# B&R Automation Studio project NAELD004C00R10L518F00 (part 9)

#### Act_OptP0200ToP0204AccDat.st
```iecst
ACTION Act_OptP0200ToP0204AccDat:

	//HComm Exchanged
	IF p_bOpsMagConvLD1HModChgDone AND p_bOpsMagConvLD2HModChgDone AND p_bOpsMagConvLD3HModChgDone THEN
		bHCommModChg := FALSE;
	END_IF

//	IF EDGENEG(p_bLFFollowerProdAccDataMnl OR p_bLCSLFAccDataMnl) THEN
//		bProdAccData	:= FALSE;
//	END_IF

	//Control
	IF (tyP0200OpsGen.tyOps.tyBtnAccDat.bRtCompl = TRUE)		OR (tyP0201OpsTravLifter.tyOps.tyBtnAccDat.bRtCompl = TRUE)
		OR (tyP0202OpsMag1.tyOps.tyBtnAccDat.bRtCompl = TRUE)	OR (tyP0203OpsMag2.tyOps.tyBtnAccDat.bRtCompl = TRUE)
		OR (tyP0204OpsMag3.tyOps.tyBtnAccDat.bRtCompl = TRUE) 	OR (tyP0206OpsMag4.tyOps.tyBtnAccDat.bRtCompl = TRUE)
		THEN

		tyP0200OpsGen.tyOps.tyBtnAccDat.bRtCompl		:= FALSE;
		tyP0201OpsTravLifter.tyOps.tyBtnAccDat.bRtCompl	:= FALSE;
		tyP0202OpsMag1.tyOps.tyBtnAccDat.bRtCompl		:= FALSE;
		tyP0203OpsMag2.tyOps.tyBtnAccDat.bRtCompl		:= FALSE;
		tyP0204OpsMag3.tyOps.tyBtnAccDat.bRtCompl		:= FALSE;
		tyP0206OpsMag4.tyOps.tyBtnAccDat.bRtCompl		:= FALSE;

		bProdAccData	:= TRUE;
	END_IF

	//Button Appearance
	IF (p_bLFFollowerProdAccDataMnl = TRUE) OR (p_bLCSLFAccDataMnl = TRUE) THEN

		fbAccDatBlinkTm(IN := TRUE);

		IF fbAccDatBlinkTm.Q THEN
			fbAccDatBlinkTm(IN := FALSE);

			IF (tyP0200OpsGen.tyOps.tyBitmapAccDat.usiValueIdx = 1) THEN
				tyP0200OpsGen.tyOps.tyBitmapAccDat.usiValueIdx			:= 0;
				tyP0201OpsTravLifter.tyOps.tyBitmapAccDat.usiValueIdx	:= 0;
				tyP0202OpsMag1.tyOps.tyBitmapAccDat.usiValueIdx			:= 0;
				tyP0203OpsMag2.tyOps.tyBitmapAccDat.usiValueIdx			:= 0;
				tyP0204OpsMag3.tyOps.tyBitmapAccDat.usiValueIdx			:= 0;
				tyP0206OpsMag4.tyOps.tyBitmapAccDat.usiValueIdx			:= 0;
			ELSE
				tyP0200OpsGen.tyOps.tyBitmapAccDat.usiValueIdx			:= 1;
				tyP0201OpsTravLifter.tyOps.tyBitmapAccDat.usiValueIdx	:= 1;
				tyP0202OpsMag1.tyOps.tyBitmapAccDat.usiValueIdx			:= 1;
				tyP0203OpsMag2.tyOps.tyBitmapAccDat.usiValueIdx			:= 1;
				tyP0204OpsMag3.tyOps.tyBitmapAccDat.usiValueIdx			:= 1;
				tyP0206OpsMag4.tyOps.tyBitmapAccDat.usiValueIdx			:= 1;
			END_IF
		END_IF

		fUIInRtStatOff(ADR(tyP0200OpsGen.tyOps.tyBtnAccDat.uiRtStat));
		fUIInRtStatOff(ADR(tyP0201OpsTravLifter.tyOps.tyBtnAccDat.uiRtStat));
		fUIInRtStatOff(ADR(tyP0202OpsMag1.tyOps.tyBtnAccDat.uiRtStat));
		fUIInRtStatOff(ADR(tyP0203OpsMag2.tyOps.tyBtnAccDat.uiRtStat));
		fUIInRtStatOff(ADR(tyP0204OpsMag3.tyOps.tyBtnAccDat.uiRtStat));
		fUIInRtStatOff(ADR(tyP0206OpsMag4.tyOps.tyBtnAccDat.uiRtStat));

		fUIInRtStatOff(ADR(tyP0200OpsGen.tyOps.tyBitmapAccDat.uiRtStat));
		fUIInRtStatOff(ADR(tyP0201OpsTravLifter.tyOps.tyBitmapAccDat.uiRtStat));
		fUIInRtStatOff(ADR(tyP0202OpsMag1.tyOps.tyBitmapAccDat.uiRtStat));
		fUIInRtStatOff(ADR(tyP0203OpsMag2.tyOps.tyBitmapAccDat.uiRtStat));
		fUIInRtStatOff(ADR(tyP0204OpsMag3.tyOps.tyBitmapAccDat.uiRtStat));
		fUIInRtStatOff(ADR(tyP0206OpsMag4.tyOps.tyBitmapAccDat.uiRtStat));
	ELSE

		fbAccDatBlinkTm(IN := FALSE);

		tyP0200OpsGen.tyOps.tyBitmapAccDat.usiValueIdx			:= 0;
		tyP0201OpsTravLifter.tyOps.tyBitmapAccDat.usiValueIdx	:= 0;
		tyP0202OpsMag1.tyOps.tyBitmapAccDat.usiValueIdx			:= 0;
		tyP0203OpsMag2.tyOps.tyBitmapAccDat.usiValueIdx			:= 0;
		tyP0204OpsMag3.tyOps.tyBitmapAccDat.usiValueIdx			:= 0;
		tyP0206OpsMag4.tyOps.tyBitmapAccDat.usiValueIdx			:= 0;

		fUIInRtStatHide(ADR(tyP0200OpsGen.tyOps.tyBtnAccDat.uiRtStat));
		fUIInRtStatHide(ADR(tyP0201OpsTravLifter.tyOps.tyBtnAccDat.uiRtStat));
		fUIInRtStatHide(ADR(tyP0202OpsMag1.tyOps.tyBtnAccDat.uiRtStat));
		fUIInRtStatHide(ADR(tyP0203OpsMag2.tyOps.tyBtnAccDat.uiRtStat));
		fUIInRtStatHide(ADR(tyP0204OpsMag3.tyOps.tyBtnAccDat.uiRtStat));
		fUIInRtStatHide(ADR(tyP0206OpsMag4.tyOps.tyBtnAccDat.uiRtStat));

		fUIInRtStatHide(ADR(tyP0200OpsGen.tyOps.tyBitmapAccDat.uiRtStat));
		fUIInRtStatHide(ADR(tyP0201OpsTravLifter.tyOps.tyBitmapAccDat.uiRtStat));
		fUIInRtStatHide(ADR(tyP0202OpsMag1.tyOps.tyBitmapAccDat.uiRtStat));
		fUIInRtStatHide(ADR(tyP0203OpsMag2.tyOps.tyBitmapAccDat.uiRtStat));
		fUIInRtStatHide(ADR(tyP0204OpsMag3.tyOps.tyBitmapAccDat.uiRtStat));
		fUIInRtStatHide(ADR(tyP0206OpsMag4.tyOps.tyBitmapAccDat.uiRtStat));
	END_IF

//	IF p_tyNtParamCurr.bLFPrep AND p_tyMcParamCurr.bLFEn THEN
//		IF p_bLFFollowerDSAllow=FALSE THEN
//			tyP0200OpsGen.tyOps.tyTxtLdrInActiveCtrl.usiValueIdx	:= 0;
//			tyP0201OpsTravLifter.tyOps.tyTxtLdrInActiveCtrl.usiValueIdx	:= 0;
//			tyP0202OpsMag1.tyOps.tyTxtLdrInActiveCtrl.usiValueIdx	:= 0;
//			tyP0203OpsMag2.tyOps.tyTxtLdrInActiveCtrl.usiValueIdx	:= 0;
//			tyP0204OpsMag3.tyOps.tyTxtLdrInActiveCtrl.usiValueIdx	:= 0;
//
//			fUIInRtStatOff(ADR(tyP0200OpsGen.tyOps.tyTxtLdrInActiveCtrl.uiRtStat));
//			fUIInRtStatOff(ADR(tyP0201OpsTravLifter.tyOps.tyTxtLdrInActiveCtrl.uiRtStat));
//			fUIInRtStatOff(ADR(tyP0202OpsMag1.tyOps.tyTxtLdrInActiveCtrl.uiRtStat));
//			fUIInRtStatOff(ADR(tyP0203OpsMag2.tyOps.tyTxtLdrInActiveCtrl.uiRtStat));
//			fUIInRtStatOff(ADR(tyP0204OpsMag3.tyOps.tyTxtLdrInActiveCtrl.uiRtStat));
//
//			fUIInRtStatOff(ADR(tyP0200OpsGen.tyOps.tyBitmapWarningLF.uiRtStat));
//			fUIInRtStatOff(ADR(tyP0201OpsTravLifter.tyOps.tyBitmapWarningLF.uiRtStat));
//			fUIInRtStatOff(ADR(tyP0202OpsMag1.tyOps.tyBitmapWarningLF.uiRtStat));
//			fUIInRtStatOff(ADR(tyP0203OpsMag2.tyOps.tyBitmapWarningLF.uiRtStat));
//			fUIInRtStatOff(ADR(tyP0204OpsMag3.tyOps.tyBitmapWarningLF.uiRtStat));
//
//		ELSIF p_bLFFollowerUSAllow=FALSE THEN
//			IF p_tyMcParamCurr.bSectionLeader THEN
//				tyP0200OpsGen.tyOps.tyTxtLdrInActiveCtrl.usiValueIdx	:= 3;
//				tyP0201OpsTravLifter.tyOps.tyTxtLdrInActiveCtrl.usiValueIdx	:= 3;
//				tyP0202OpsMag1.tyOps.tyTxtLdrInActiveCtrl.usiValueIdx	:= 3;
//				tyP0203OpsMag2.tyOps.tyTxtLdrInActiveCtrl.usiValueIdx	:= 3;
//				tyP0204OpsMag3.tyOps.tyTxtLdrInActiveCtrl.usiValueIdx	:= 3;
//
//				fUIInRtStatOff(ADR(tyP0200OpsGen.tyOps.tyTxtLdrInActiveCtrl.uiRtStat));
//				fUIInRtStatOff(ADR(tyP0201OpsTravLifter.tyOps.tyTxtLdrInActiveCtrl.uiRtStat));
//				fUIInRtStatOff(ADR(tyP0202OpsMag1.tyOps.tyTxtLdrInActiveCtrl.uiRtStat));
//				fUIInRtStatOff(ADR(tyP0203OpsMag2.tyOps.tyTxtLdrInActiveCtrl.uiRtStat));
//				fUIInRtStatOff(ADR(tyP0204OpsMag3.tyOps.tyTxtLdrInActiveCtrl.uiRtStat));
//
//				fUIInRtStatOff(ADR(tyP0200OpsGen.tyOps.tyBitmapWarningLF.uiRtStat));
//				fUIInRtStatOff(ADR(tyP0201OpsTravLifter.tyOps.tyBitmapWarningLF.uiRtStat));
//				fUIInRtStatOff(ADR(tyP0202OpsMag1.tyOps.tyBitmapWarningLF.uiRtStat));
//				fUIInRtStatOff(ADR(tyP0203OpsMag2.tyOps.tyBitmapWarningLF.uiRtStat));
//				fUIInRtStatOff(ADR(tyP0204OpsMag3.tyOps.tyBitmapWarningLF.uiRtStat));
//			ELSE
//				tyP0200OpsGen.tyOps.tyTxtLdrInActiveCtrl.usiValueIdx	:= 2;
//				tyP0201OpsTravLifter.tyOps.tyTxtLdrInActiveCtrl.usiValueIdx	:= 2;
//				tyP0202OpsMag1.tyOps.tyTxtLdrInActiveCtrl.usiValueIdx	:= 2;
//				tyP0203OpsMag2.tyOps.tyTxtLdrInActiveCtrl.usiValueIdx	:= 2;
//				tyP0204OpsMag3.tyOps.tyTxtLdrInActiveCtrl.usiValueIdx	:= 2;
//
//				fUIInRtStatOff(ADR(tyP0200OpsGen.tyOps.tyTxtLdrInActiveCtrl.uiRtStat));
//				fUIInRtStatOff(ADR(tyP0201OpsTravLifter.tyOps.tyTxtLdrInActiveCtrl.uiRtStat));
//				fUIInRtStatOff(ADR(tyP0202OpsMag1.tyOps.tyTxtLdrInActiveCtrl.uiRtStat));
//				fUIInRtStatOff(ADR(tyP0203OpsMag2.tyOps.tyTxtLdrInActiveCtrl.uiRtStat));
//				fUIInRtStatOff(ADR(tyP0204OpsMag3.tyOps.tyTxtLdrInActiveCtrl.uiRtStat));
//
//				fUIInRtStatOff(ADR(tyP0200OpsGen.tyOps.tyBitmapWarningLF.uiRtStat));
//				fUIInRtStatOff(ADR(tyP0201OpsTravLifter.tyOps.tyBitmapWarningLF.uiRtStat));
//				fUIInRtStatOff(ADR(tyP0202OpsMag1.tyOps.tyBitmapWarningLF.uiRtStat));
//				fUIInRtStatOff(ADR(tyP0203OpsMag2.tyOps.tyBitmapWarningLF.uiRtStat));
//				fUIInRtStatOff(ADR(tyP0204OpsMag3.tyOps.tyBitmapWarningLF.uiRtStat));
//			END_IF
//		ELSE
//			IF p_bLFFollowerLdrSeqCtrlInActive THEN
//				tyP0200OpsGen.tyOps.tyTxtLdrInActiveCtrl.usiValueIdx	:= 1;
//				tyP0201OpsTravLifter.tyOps.tyTxtLdrInActiveCtrl.usiValueIdx	:= 1;
//				tyP0202OpsMag1.tyOps.tyTxtLdrInActiveCtrl.usiValueIdx	:= 1;
//				tyP0203OpsMag2.tyOps.tyTxtLdrInActiveCtrl.usiValueIdx	:= 1;
//				tyP0204OpsMag3.tyOps.tyTxtLdrInActiveCtrl.usiValueIdx	:= 1;
//
//				fUIInRtStatOff(ADR(tyP0200OpsGen.tyOps.tyTxtLdrInActiveCtrl.uiRtStat));
//				fUIInRtStatOff(ADR(tyP0201OpsTravLifter.tyOps.tyTxtLdrInActiveCtrl.uiRtStat));
//				fUIInRtStatOff(ADR(tyP0202OpsMag1.tyOps.tyTxtLdrInActiveCtrl.uiRtStat));
//				fUIInRtStatOff(ADR(tyP0203OpsMag2.tyOps.tyTxtLdrInActiveCtrl.uiRtStat));
//				fUIInRtStatOff(ADR(tyP0204OpsMag3.tyOps.tyTxtLdrInActiveCtrl.uiRtStat));
//
//				fUIInRtStatOff(ADR(tyP0200OpsGen.tyOps.tyBitmapWarningLF.uiRtStat));
//				fUIInRtStatOff(ADR(tyP0201OpsTravLifter.tyOps.tyBitmapWarningLF.uiRtStat));
//				fUIInRtStatOff(ADR(tyP0202OpsMag1.tyOps.tyBitmapWarningLF.uiRtStat));
//				fUIInRtStatOff(ADR(tyP0203OpsMag2.tyOps.tyBitmapWarningLF.uiRtStat));
//				fUIInRtStatOff(ADR(tyP0204OpsMag3.tyOps.tyBitmapWarningLF.uiRtStat));
//			ELSE
//				fUIInRtStatHide(ADR(tyP0200OpsGen.tyOps.tyTxtLdrInActiveCtrl.uiRtStat));
//				fUIInRtStatHide(ADR(tyP0201OpsTravLifter.tyOps.tyTxtLdrInActiveCtrl.uiRtStat));
//				fUIInRtStatHide(ADR(tyP0202OpsMag1.tyOps.tyTxtLdrInActiveCtrl.uiRtStat));
//				fUIInRtStatHide(ADR(tyP0203OpsMag2.tyOps.tyTxtLdrInActiveCtrl.uiRtStat));
//				fUIInRtStatHide(ADR(tyP0204OpsMag3.tyOps.tyTxtLdrInActiveCtrl.uiRtStat));
//
//				fUIInRtStatHide(ADR(tyP0200OpsGen.tyOps.tyBitmapWarningLF.uiRtStat));
//				fUIInRtStatHide(ADR(tyP0201OpsTravLifter.tyOps.tyBitmapWarningLF.uiRtStat));
//				fUIInRtStatHide(ADR(tyP0202OpsMag1.tyOps.tyBitmapWarningLF.uiRtStat));
//				fUIInRtStatHide(ADR(tyP0203OpsMag2.tyOps.tyBitmapWarningLF.uiRtStat));
//				fUIInRtStatHide(ADR(tyP0204OpsMag3.tyOps.tyBitmapWarningLF.uiRtStat));
//			END_IF
//		END_IF
//	ELSE
//		fUIInRtStatHide(ADR(tyP0200OpsGen.tyOps.tyTxtLdrInActiveCtrl.uiRtStat));
//		fUIInRtStatHide(ADR(tyP0201OpsTravLifter.tyOps.tyTxtLdrInActiveCtrl.uiRtStat));
//		fUIInRtStatHide(ADR(tyP0202OpsMag1.tyOps.tyTxtLdrInActiveCtrl.uiRtStat));
//		fUIInRtStatHide(ADR(tyP0203OpsMag2.tyOps.tyTxtLdrInActiveCtrl.uiRtStat));
//		fUIInRtStatHide(ADR(tyP0204OpsMag3.tyOps.tyTxtLdrInActiveCtrl.uiRtStat));
//
//		fUIInRtStatHide(ADR(tyP0200OpsGen.tyOps.tyBitmapWarningLF.uiRtStat));
//		fUIInRtStatHide(ADR(tyP0201OpsTravLifter.tyOps.tyBitmapWarningLF.uiRtStat));
//		fUIInRtStatHide(ADR(tyP0202OpsMag1.tyOps.tyBitmapWarningLF.uiRtStat));
//		fUIInRtStatHide(ADR(tyP0203OpsMag2.tyOps.tyBitmapWarningLF.uiRtStat));
//		fUIInRtStatHide(ADR(tyP0204OpsMag3.tyOps.tyBitmapWarningLF.uiRtStat));
//	END_IF

END_ACTION
```

#### Act_OptP0200ToP0204BypsInitConv.st
```iecst
ACTION Act_OptP0200ToP0204BypsInitConv:

	IF p_tyNtParamCurr.bProjBypsInitConvPrep THEN

		(*Display*)
		//Initializing Conveyor
		IF EDGEPOS(p_bOpsTravLifLDInitConv) THEN
			fUIInRtStatOff(ADR(tyP0200OpsGen.tyBypsInitConv.tyLyr.uiRtStat));
			fUIInRtStatOff(ADR(tyP0201OpsTravLifter.tyBypsInitConv.tyLyr.uiRtStat));
			fUIInRtStatOff(ADR(tyP0202OpsMag1.tyBypsInitConv.tyLyr.uiRtStat));
			fUIInRtStatOff(ADR(tyP0203OpsMag2.tyBypsInitConv.tyLyr.uiRtStat));
			fUIInRtStatOff(ADR(tyP0204OpsMag3.tyBypsInitConv.tyLyr.uiRtStat));
			fUIInRtStatOff(ADR(tyP0206OpsMag4.tyBypsInitConv.tyLyr.uiRtStat));
		END_IF

		//Initializing Conveyor Done
		IF EDGENEG(p_bOpsTravLifLDInitConv) THEN
			fUIInRtStatHide(ADR(tyP0200OpsGen.tyBypsInitConv.tyLyr.uiRtStat));
			fUIInRtStatHide(ADR(tyP0201OpsTravLifter.tyBypsInitConv.tyLyr.uiRtStat));
			fUIInRtStatHide(ADR(tyP0202OpsMag1.tyBypsInitConv.tyLyr.uiRtStat));
			fUIInRtStatHide(ADR(tyP0203OpsMag2.tyBypsInitConv.tyLyr.uiRtStat));
			fUIInRtStatHide(ADR(tyP0204OpsMag3.tyBypsInitConv.tyLyr.uiRtStat));
			fUIInRtStatHide(ADR(tyP0206OpsMag4.tyBypsInitConv.tyLyr.uiRtStat));

			bOpsBypsInitConv	:= FALSE;
		END_IF

		//Blinking Button
		IF tyP0200OpsGen.tyBypsInitConv.tyLyr.uiRtStat.0 = FALSE THEN

			fbBypsInitConvBlinkTm(IN := TRUE);

			IF fbBypsInitConvBlinkTm.Q THEN
				fbBypsInitConvBlinkTm(IN := FALSE);

				IF tyP0200OpsGen.tyBypsInitConv.tyBtnBypsInitConv.usiBitmapIdx = 0 THEN
					tyP0200OpsGen.tyBypsInitConv.tyBtnBypsInitConv.usiBitmapIdx			:= 1;
					tyP0201OpsTravLifter.tyBypsInitConv.tyBtnBypsInitConv.usiBitmapIdx	:= 1;
					tyP0202OpsMag1.tyBypsInitConv.tyBtnBypsInitConv.usiBitmapIdx		:= 1;
					tyP0203OpsMag2.tyBypsInitConv.tyBtnBypsInitConv.usiBitmapIdx		:= 1;
					tyP0204OpsMag3.tyBypsInitConv.tyBtnBypsInitConv.usiBitmapIdx		:= 1;
					tyP0206OpsMag4.tyBypsInitConv.tyBtnBypsInitConv.usiBitmapIdx		:= 1;
				ELSE
					tyP0200OpsGen.tyBypsInitConv.tyBtnBypsInitConv.usiBitmapIdx			:= 0;
					tyP0201OpsTravLifter.tyBypsInitConv.tyBtnBypsInitConv.usiBitmapIdx	:= 0;
					tyP0202OpsMag1.tyBypsInitConv.tyBtnBypsInitConv.usiBitmapIdx		:= 0;
					tyP0203OpsMag2.tyBypsInitConv.tyBtnBypsInitConv.usiBitmapIdx		:= 0;
					tyP0204OpsMag3.tyBypsInitConv.tyBtnBypsInitConv.usiBitmapIdx		:= 0;
					tyP0206OpsMag4.tyBypsInitConv.tyBtnBypsInitConv.usiBitmapIdx		:= 0;
				END_IF

			END_IF

		ELSE

			fbBypsInitConvBlinkTm(IN := FALSE);

			tyP0200OpsGen.tyBypsInitConv.tyBtnBypsInitConv.usiBitmapIdx			:= 0;
			tyP0201OpsTravLifter.tyBypsInitConv.tyBtnBypsInitConv.usiBitmapIdx	:= 0;
			tyP0202OpsMag1.tyBypsInitConv.tyBtnBypsInitConv.usiBitmapIdx		:= 0;
			tyP0203OpsMag2.tyBypsInitConv.tyBtnBypsInitConv.usiBitmapIdx		:= 0;
			tyP0204OpsMag3.tyBypsInitConv.tyBtnBypsInitConv.usiBitmapIdx		:= 0;
			tyP0206OpsMag4.tyBypsInitConv.tyBtnBypsInitConv.usiBitmapIdx		:= 0;
		END_IF

		(*Control*)
		IF tyP0200OpsGen.tyBypsInitConv.tyBtnBypsInitConv.bRtCompl
			OR tyP0201OpsTravLifter.tyBypsInitConv.tyBtnBypsInitConv.bRtCompl
			OR tyP0202OpsMag1.tyBypsInitConv.tyBtnBypsInitConv.bRtCompl
			OR tyP0203OpsMag2.tyBypsInitConv.tyBtnBypsInitConv.bRtCompl
			OR tyP0204OpsMag3.tyBypsInitConv.tyBtnBypsInitConv.bRtCompl
			OR tyP0206OpsMag4.tyBypsInitConv.tyBtnBypsInitConv.bRtCompl
			THEN
			tyP0200OpsGen.tyBypsInitConv.tyBtnBypsInitConv.bRtCompl			:= FALSE;
			tyP0201OpsTravLifter.tyBypsInitConv.tyBtnBypsInitConv.bRtCompl	:= FALSE;
			tyP0202OpsMag1.tyBypsInitConv.tyBtnBypsInitConv.bRtCompl		:= FALSE;
			tyP0203OpsMag2.tyBypsInitConv.tyBtnBypsInitConv.bRtCompl		:= FALSE;
			tyP0204OpsMag3.tyBypsInitConv.tyBtnBypsInitConv.bRtCompl		:= FALSE;
			tyP0206OpsMag4.tyBypsInitConv.tyBtnBypsInitConv.bRtCompl		:= FALSE;

			fUIInRtStatHide(ADR(tyP0200OpsGen.tyBypsInitConv.tyLyr.uiRtStat));
			fUIInRtStatHide(ADR(tyP0201OpsTravLifter.tyBypsInitConv.tyLyr.uiRtStat));
			fUIInRtStatHide(ADR(tyP0202OpsMag1.tyBypsInitConv.tyLyr.uiRtStat));
			fUIInRtStatHide(ADR(tyP0203OpsMag2.tyBypsInitConv.tyLyr.uiRtStat));
			fUIInRtStatHide(ADR(tyP0204OpsMag3.tyBypsInitConv.tyLyr.uiRtStat));
			fUIInRtStatHide(ADR(tyP0206OpsMag4.tyBypsInitConv.tyLyr.uiRtStat));
			bOpsBypsInitConv	:= TRUE;

		ELSIF tyP0200OpsGen.tyBypsInitConv.tyHotspotClose.bRtCompl
			OR tyP0201OpsTravLifter.tyBypsInitConv.tyHotspotClose.bRtCompl
			OR tyP0202OpsMag1.tyBypsInitConv.tyHotspotClose.bRtCompl
			OR tyP0203OpsMag2.tyBypsInitConv.tyHotspotClose.bRtCompl
			OR tyP0204OpsMag3.tyBypsInitConv.tyHotspotClose.bRtCompl
			OR tyP0206OpsMag4.tyBypsInitConv.tyHotspotClose.bRtCompl
			THEN
			tyP0200OpsGen.tyBypsInitConv.tyHotspotClose.bRtCompl		:= FALSE;
			tyP0201OpsTravLifter.tyBypsInitConv.tyHotspotClose.bRtCompl	:= FALSE;
			tyP0202OpsMag1.tyBypsInitConv.tyHotspotClose.bRtCompl		:= FALSE;
			tyP0203OpsMag2.tyBypsInitConv.tyHotspotClose.bRtCompl		:= FALSE;
			tyP0204OpsMag3.tyBypsInitConv.tyHotspotClose.bRtCompl		:= FALSE;
			tyP0206OpsMag4.tyBypsInitConv.tyHotspotClose.bRtCompl		:= FALSE;

			fUIInRtStatHide(ADR(tyP0200OpsGen.tyBypsInitConv.tyLyr.uiRtStat));
			fUIInRtStatHide(ADR(tyP0201OpsTravLifter.tyBypsInitConv.tyLyr.uiRtStat));
			fUIInRtStatHide(ADR(tyP0202OpsMag1.tyBypsInitConv.tyLyr.uiRtStat));
			fUIInRtStatHide(ADR(tyP0203OpsMag2.tyBypsInitConv.tyLyr.uiRtStat));
			fUIInRtStatHide(ADR(tyP0204OpsMag3.tyBypsInitConv.tyLyr.uiRtStat));
			fUIInRtStatHide(ADR(tyP0206OpsMag4.tyBypsInitConv.tyLyr.uiRtStat));
		END_IF

	END_IF

END_ACTION
```

#### Act_OptP0200ToP0204_P0003AccDat.st - not listed in the package file held
```iecst
ACTION Act_OptP0200ToP0204_P0003AccDat:

	//HComm Exchanged
	IF p_bOpsMagConvLD1HModChgDone AND p_bOpsMagConvLD2HModChgDone AND p_bOpsMagConvLD3HModChgDone THEN
		bHCommModChg := FALSE;
	END_IF

//	IF EDGENEG(p_bLFFollowerProdAccDataMnl OR p_bLCSLFAccDataMnl) THEN
//		bProdAccData	:= FALSE;
//	END_IF

	//Control
	IF (tyP0200OpsGen.tyOps.tyBtnAccDat.bRtCompl = TRUE)		OR (tyP0201OpsTravLifter.tyOps.tyBtnAccDat.bRtCompl = TRUE)
		OR (tyP0202OpsMag1.tyOps.tyBtnAccDat.bRtCompl = TRUE)	OR (tyP0203OpsMag2.tyOps.tyBtnAccDat.bRtCompl = TRUE)
		OR (tyP0204OpsMag3.tyOps.tyBtnAccDat.bRtCompl = TRUE) 	OR (tyP0206OpsMag4.tyOps.tyBtnAccDat.bRtCompl = TRUE)
		OR tyP0003MMenu.tyMMenuBtn.tyBtnAccDat.bRtCompl THEN

		tyP0200OpsGen.tyOps.tyBtnAccDat.bRtCompl		:= FALSE;
		tyP0201OpsTravLifter.tyOps.tyBtnAccDat.bRtCompl	:= FALSE;
		tyP0202OpsMag1.tyOps.tyBtnAccDat.bRtCompl		:= FALSE;
		tyP0203OpsMag2.tyOps.tyBtnAccDat.bRtCompl		:= FALSE;
		tyP0204OpsMag3.tyOps.tyBtnAccDat.bRtCompl		:= FALSE;
		tyP0206OpsMag4.tyOps.tyBtnAccDat.bRtCompl		:= FALSE;
		tyP0003MMenu.tyMMenuBtn.tyBtnAccDat.bRtCompl := FALSE;

		bProdAccData	:= TRUE;
	END_IF

	//Button Appearance
	IF (p_bLFFollowerProdAccDataMnl = TRUE) OR (p_bLCSLFAccDataMnl = TRUE) THEN

		fbAccDatBlinkTm(IN := TRUE);

		IF fbAccDatBlinkTm.Q THEN
			fbAccDatBlinkTm(IN := FALSE);

			IF (tyP0200OpsGen.tyOps.tyBitmapAccDat.usiValueIdx = 1) THEN
				tyP0200OpsGen.tyOps.tyBitmapAccDat.usiValueIdx			:= 0;
				tyP0201OpsTravLifter.tyOps.tyBitmapAccDat.usiValueIdx	:= 0;
				tyP0202OpsMag1.tyOps.tyBitmapAccDat.usiValueIdx			:= 0;
				tyP0203OpsMag2.tyOps.tyBitmapAccDat.usiValueIdx			:= 0;
				tyP0204OpsMag3.tyOps.tyBitmapAccDat.usiValueIdx			:= 0;
				tyP0206OpsMag4.tyOps.tyBitmapAccDat.usiValueIdx			:= 0;
				tyP0003MMenu.tyMMenuBtn.tyBtnAccDat.usiBitmapIdx := 0;
			ELSE
				tyP0200OpsGen.tyOps.tyBitmapAccDat.usiValueIdx			:= 1;
				tyP0201OpsTravLifter.tyOps.tyBitmapAccDat.usiValueIdx	:= 1;
				tyP0202OpsMag1.tyOps.tyBitmapAccDat.usiValueIdx			:= 1;
				tyP0203OpsMag2.tyOps.tyBitmapAccDat.usiValueIdx			:= 1;
				tyP0204OpsMag3.tyOps.tyBitmapAccDat.usiValueIdx			:= 1;
				tyP0206OpsMag4.tyOps.tyBitmapAccDat.usiValueIdx			:= 1;
				tyP0003MMenu.tyMMenuBtn.tyBtnAccDat.usiBitmapIdx := 4;
			END_IF
		END_IF

		fUIInRtStatOff(ADR(tyP0200OpsGen.tyOps.tyBtnAccDat.uiRtStat));
		fUIInRtStatOff(ADR(tyP0201OpsTravLifter.tyOps.tyBtnAccDat.uiRtStat));
		fUIInRtStatOff(ADR(tyP0202OpsMag1.tyOps.tyBtnAccDat.uiRtStat));
		fUIInRtStatOff(ADR(tyP0203OpsMag2.tyOps.tyBtnAccDat.uiRtStat));
		fUIInRtStatOff(ADR(tyP0204OpsMag3.tyOps.tyBtnAccDat.uiRtStat));
		fUIInRtStatOff(ADR(tyP0206OpsMag4.tyOps.tyBtnAccDat.uiRtStat));

		fUIInRtStatOff(ADR(tyP0200OpsGen.tyOps.tyBitmapAccDat.uiRtStat));
		fUIInRtStatOff(ADR(tyP0201OpsTravLifter.tyOps.tyBitmapAccDat.uiRtStat));
		fUIInRtStatOff(ADR(tyP0202OpsMag1.tyOps.tyBitmapAccDat.uiRtStat));
		fUIInRtStatOff(ADR(tyP0203OpsMag2.tyOps.tyBitmapAccDat.uiRtStat));
		fUIInRtStatOff(ADR(tyP0204OpsMag3.tyOps.tyBitmapAccDat.uiRtStat));
		fUIInRtStatOff(ADR(tyP0206OpsMag4.tyOps.tyBitmapAccDat.uiRtStat));

		fUIInRtStatOff(ADR(tyP0003MMenu.tyMMenuBtn.tyBtnAccDat.uiRtStat));
	ELSE

		fbAccDatBlinkTm(IN := FALSE);

		tyP0200OpsGen.tyOps.tyBitmapAccDat.usiValueIdx			:= 0;
		tyP0201OpsTravLifter.tyOps.tyBitmapAccDat.usiValueIdx	:= 0;
		tyP0202OpsMag1.tyOps.tyBitmapAccDat.usiValueIdx			:= 0;
		tyP0203OpsMag2.tyOps.tyBitmapAccDat.usiValueIdx			:= 0;
		tyP0204OpsMag3.tyOps.tyBitmapAccDat.usiValueIdx			:= 0;
		tyP0206OpsMag4.tyOps.tyBitmapAccDat.usiValueIdx			:= 0;

		fUIInRtStatHide(ADR(tyP0200OpsGen.tyOps.tyBtnAccDat.uiRtStat));
		fUIInRtStatHide(ADR(tyP0201OpsTravLifter.tyOps.tyBtnAccDat.uiRtStat));
		fUIInRtStatHide(ADR(tyP0202OpsMag1.tyOps.tyBtnAccDat.uiRtStat));
		fUIInRtStatHide(ADR(tyP0203OpsMag2.tyOps.tyBtnAccDat.uiRtStat));
		fUIInRtStatHide(ADR(tyP0204OpsMag3.tyOps.tyBtnAccDat.uiRtStat));
		fUIInRtStatHide(ADR(tyP0206OpsMag4.tyOps.tyBtnAccDat.uiRtStat));

		fUIInRtStatHide(ADR(tyP0200OpsGen.tyOps.tyBitmapAccDat.uiRtStat));
		fUIInRtStatHide(ADR(tyP0201OpsTravLifter.tyOps.tyBitmapAccDat.uiRtStat));
		fUIInRtStatHide(ADR(tyP0202OpsMag1.tyOps.tyBitmapAccDat.uiRtStat));
		fUIInRtStatHide(ADR(tyP0203OpsMag2.tyOps.tyBitmapAccDat.uiRtStat));
		fUIInRtStatHide(ADR(tyP0204OpsMag3.tyOps.tyBitmapAccDat.uiRtStat));
		fUIInRtStatHide(ADR(tyP0206OpsMag4.tyOps.tyBitmapAccDat.uiRtStat));

		fUIInRtStatHide(ADR(tyP0003MMenu.tyMMenuBtn.tyBtnAccDat.uiRtStat));
	END_IF

//	IF p_tyNtParamCurr.bLFPrep AND p_tyMcParamCurr.bLFEn THEN
//		IF p_bLFFollowerDSAllow=FALSE THEN
//			tyP0200OpsGen.tyOps.tyTxtLdrInActiveCtrl.usiValueIdx	:= 0;
//			tyP0201OpsTravLifter.tyOps.tyTxtLdrInActiveCtrl.usiValueIdx	:= 0;
//			tyP0202OpsMag1.tyOps.tyTxtLdrInActiveCtrl.usiValueIdx	:= 0;
//			tyP0203OpsMag2.tyOps.tyTxtLdrInActiveCtrl.usiValueIdx	:= 0;
//			tyP0204OpsMag3.tyOps.tyTxtLdrInActiveCtrl.usiValueIdx	:= 0;
//
//			fUIInRtStatOff(ADR(tyP0200OpsGen.tyOps.tyTxtLdrInActiveCtrl.uiRtStat));
//			fUIInRtStatOff(ADR(tyP0201OpsTravLifter.tyOps.tyTxtLdrInActiveCtrl.uiRtStat));
//			fUIInRtStatOff(ADR(tyP0202OpsMag1.tyOps.tyTxtLdrInActiveCtrl.uiRtStat));
//			fUIInRtStatOff(ADR(tyP0203OpsMag2.tyOps.tyTxtLdrInActiveCtrl.uiRtStat));
//			fUIInRtStatOff(ADR(tyP0204OpsMag3.tyOps.tyTxtLdrInActiveCtrl.uiRtStat));
//
//			fUIInRtStatOff(ADR(tyP0200OpsGen.tyOps.tyBitmapWarningLF.uiRtStat));
//			fUIInRtStatOff(ADR(tyP0201OpsTravLifter.tyOps.tyBitmapWarningLF.uiRtStat));
//			fUIInRtStatOff(ADR(tyP0202OpsMag1.tyOps.tyBitmapWarningLF.uiRtStat));
//			fUIInRtStatOff(ADR(tyP0203OpsMag2.tyOps.tyBitmapWarningLF.uiRtStat));
//			fUIInRtStatOff(ADR(tyP0204OpsMag3.tyOps.tyBitmapWarningLF.uiRtStat));
//
//		ELSIF p_bLFFollowerUSAllow=FALSE THEN
//			IF p_tyMcParamCurr.bSectionLeader THEN
//				tyP0200OpsGen.tyOps.tyTxtLdrInActiveCtrl.usiValueIdx	:= 3;
//				tyP0201OpsTravLifter.tyOps.tyTxtLdrInActiveCtrl.usiValueIdx	:= 3;
//				tyP0202OpsMag1.tyOps.tyTxtLdrInActiveCtrl.usiValueIdx	:= 3;
//				tyP0203OpsMag2.tyOps.tyTxtLdrInActiveCtrl.usiValueIdx	:= 3;
//				tyP0204OpsMag3.tyOps.tyTxtLdrInActiveCtrl.usiValueIdx	:= 3;
//
//				fUIInRtStatOff(ADR(tyP0200OpsGen.tyOps.tyTxtLdrInActiveCtrl.uiRtStat));
//				fUIInRtStatOff(ADR(tyP0201OpsTravLifter.tyOps.tyTxtLdrInActiveCtrl.uiRtStat));
//				fUIInRtStatOff(ADR(tyP0202OpsMag1.tyOps.tyTxtLdrInActiveCtrl.uiRtStat));
//				fUIInRtStatOff(ADR(tyP0203OpsMag2.tyOps.tyTxtLdrInActiveCtrl.uiRtStat));
//				fUIInRtStatOff(ADR(tyP0204OpsMag3.tyOps.tyTxtLdrInActiveCtrl.uiRtStat));
//
//				fUIInRtStatOff(ADR(tyP0200OpsGen.tyOps.tyBitmapWarningLF.uiRtStat));
//				fUIInRtStatOff(ADR(tyP0201OpsTravLifter.tyOps.tyBitmapWarningLF.uiRtStat));
//				fUIInRtStatOff(ADR(tyP0202OpsMag1.tyOps.tyBitmapWarningLF.uiRtStat));
//				fUIInRtStatOff(ADR(tyP0203OpsMag2.tyOps.tyBitmapWarningLF.uiRtStat));
//				fUIInRtStatOff(ADR(tyP0204OpsMag3.tyOps.tyBitmapWarningLF.uiRtStat));
//			ELSE
//				tyP0200OpsGen.tyOps.tyTxtLdrInActiveCtrl.usiValueIdx	:= 2;
//				tyP0201OpsTravLifter.tyOps.tyTxtLdrInActiveCtrl.usiValueIdx	:= 2;
//				tyP0202OpsMag1.tyOps.tyTxtLdrInActiveCtrl.usiValueIdx	:= 2;
//				tyP0203OpsMag2.tyOps.tyTxtLdrInActiveCtrl.usiValueIdx	:= 2;
//				tyP0204OpsMag3.tyOps.tyTxtLdrInActiveCtrl.usiValueIdx	:= 2;
//
//				fUIInRtStatOff(ADR(tyP0200OpsGen.tyOps.tyTxtLdrInActiveCtrl.uiRtStat));
//				fUIInRtStatOff(ADR(tyP0201OpsTravLifter.tyOps.tyTxtLdrInActiveCtrl.uiRtStat));
//				fUIInRtStatOff(ADR(tyP0202OpsMag1.tyOps.tyTxtLdrInActiveCtrl.uiRtStat));
//				fUIInRtStatOff(ADR(tyP0203OpsMag2.tyOps.tyTxtLdrInActiveCtrl.uiRtStat));
//				fUIInRtStatOff(ADR(tyP0204OpsMag3.tyOps.tyTxtLdrInActiveCtrl.uiRtStat));
//
//				fUIInRtStatOff(ADR(tyP0200OpsGen.tyOps.tyBitmapWarningLF.uiRtStat));
//				fUIInRtStatOff(ADR(tyP0201OpsTravLifter.tyOps.tyBitmapWarningLF.uiRtStat));
//				fUIInRtStatOff(ADR(tyP0202OpsMag1.tyOps.tyBitmapWarningLF.uiRtStat));
//				fUIInRtStatOff(ADR(tyP0203OpsMag2.tyOps.tyBitmapWarningLF.uiRtStat));
//				fUIInRtStatOff(ADR(tyP0204OpsMag3.tyOps.tyBitmapWarningLF.uiRtStat));
//			END_IF
//		ELSE
//			IF p_bLFFollowerLdrSeqCtrlInActive THEN
//				tyP0200OpsGen.tyOps.tyTxtLdrInActiveCtrl.usiValueIdx	:= 1;
//				tyP0201OpsTravLifter.tyOps.tyTxtLdrInActiveCtrl.usiValueIdx	:= 1;
//				tyP0202OpsMag1.tyOps.tyTxtLdrInActiveCtrl.usiValueIdx	:= 1;
//				tyP0203OpsMag2.tyOps.tyTxtLdrInActiveCtrl.usiValueIdx	:= 1;
//				tyP0204OpsMag3.tyOps.tyTxtLdrInActiveCtrl.usiValueIdx	:= 1;
//
//				fUIInRtStatOff(ADR(tyP0200OpsGen.tyOps.tyTxtLdrInActiveCtrl.uiRtStat));
//				fUIInRtStatOff(ADR(tyP0201OpsTravLifter.tyOps.tyTxtLdrInActiveCtrl.uiRtStat));
//				fUIInRtStatOff(ADR(tyP0202OpsMag1.tyOps.tyTxtLdrInActiveCtrl.uiRtStat));
//				fUIInRtStatOff(ADR(tyP0203OpsMag2.tyOps.tyTxtLdrInActiveCtrl.uiRtStat));
//				fUIInRtStatOff(ADR(tyP0204OpsMag3.tyOps.tyTxtLdrInActiveCtrl.uiRtStat));
//
//				fUIInRtStatOff(ADR(tyP0200OpsGen.tyOps.tyBitmapWarningLF.uiRtStat));
//				fUIInRtStatOff(ADR(tyP0201OpsTravLifter.tyOps.tyBitmapWarningLF.uiRtStat));
//				fUIInRtStatOff(ADR(tyP0202OpsMag1.tyOps.tyBitmapWarningLF.uiRtStat));
//				fUIInRtStatOff(ADR(tyP0203OpsMag2.tyOps.tyBitmapWarningLF.uiRtStat));
//				fUIInRtStatOff(ADR(tyP0204OpsMag3.tyOps.tyBitmapWarningLF.uiRtStat));
//			ELSE
//				fUIInRtStatHide(ADR(tyP0200OpsGen.tyOps.tyTxtLdrInActiveCtrl.uiRtStat));
//				fUIInRtStatHide(ADR(tyP0201OpsTravLifter.tyOps.tyTxtLdrInActiveCtrl.uiRtStat));
//				fUIInRtStatHide(ADR(tyP0202OpsMag1.tyOps.tyTxtLdrInActiveCtrl.uiRtStat));
//				fUIInRtStatHide(ADR(tyP0203OpsMag2.tyOps.tyTxtLdrInActiveCtrl.uiRtStat));
//				fUIInRtStatHide(ADR(tyP0204OpsMag3.tyOps.tyTxtLdrInActiveCtrl.uiRtStat));
//
//				fUIInRtStatHide(ADR(tyP0200OpsGen.tyOps.tyBitmapWarningLF.uiRtStat));
//				fUIInRtStatHide(ADR(tyP0201OpsTravLifter.tyOps.tyBitmapWarningLF.uiRtStat));
//				fUIInRtStatHide(ADR(tyP0202OpsMag1.tyOps.tyBitmapWarningLF.uiRtStat));
//				fUIInRtStatHide(ADR(tyP0203OpsMag2.tyOps.tyBitmapWarningLF.uiRtStat));
//				fUIInRtStatHide(ADR(tyP0204OpsMag3.tyOps.tyBitmapWarningLF.uiRtStat));
//			END_IF
//		END_IF
//	ELSE
//		fUIInRtStatHide(ADR(tyP0200OpsGen.tyOps.tyTxtLdrInActiveCtrl.uiRtStat));
//		fUIInRtStatHide(ADR(tyP0201OpsTravLifter.tyOps.tyTxtLdrInActiveCtrl.uiRtStat));
//		fUIInRtStatHide(ADR(tyP0202OpsMag1.tyOps.tyTxtLdrInActiveCtrl.uiRtStat));
//		fUIInRtStatHide(ADR(tyP0203OpsMag2.tyOps.tyTxtLdrInActiveCtrl.uiRtStat));
//		fUIInRtStatHide(ADR(tyP0204OpsMag3.tyOps.tyTxtLdrInActiveCtrl.uiRtStat));
//
//		fUIInRtStatHide(ADR(tyP0200OpsGen.tyOps.tyBitmapWarningLF.uiRtStat));
//		fUIInRtStatHide(ADR(tyP0201OpsTravLifter.tyOps.tyBitmapWarningLF.uiRtStat));
//		fUIInRtStatHide(ADR(tyP0202OpsMag1.tyOps.tyBitmapWarningLF.uiRtStat));
//		fUIInRtStatHide(ADR(tyP0203OpsMag2.tyOps.tyBitmapWarningLF.uiRtStat));
//		fUIInRtStatHide(ADR(tyP0204OpsMag3.tyOps.tyBitmapWarningLF.uiRtStat));
//	END_IF

END_ACTION
```

#### Act_OptP0202ToP0204UnloadMag.st
```iecst
ACTION Act_OptP0202ToP0204UnloadMag:

	//Reset
	IF EDGEPOS(p_bOpsStatusStop) THEN
		bUnloadMag	:= FALSE;

		tyP0202OpsMag1.tyOps.tyBtnUnloadMag.bRtCompl	:= FALSE;
		tyP0203OpsMag2.tyOps.tyBtnUnloadMag.bRtCompl	:= FALSE;
		tyP0204OpsMag3.tyOps.tyBtnUnloadMag.bRtCompl	:= FALSE;

		p_tyC0008MsgBox ACCESS ADR(tyP0202OpsMag1.tyMsgBoxHide);
		p_tyC0008MsgBox ACCESS ADR(tyP0203OpsMag2.tyMsgBoxHide);
		p_tyC0008MsgBox ACCESS ADR(tyP0204OpsMag3.tyMsgBoxHide);
	END_IF

	//Control
	IF tyP0202OpsMag1.tyOps.tyBtnUnloadMag.bRtCompl = TRUE THEN

		IF bUnloadMag = FALSE THEN

			p_tyC0008MsgBox ACCESS ADR(tyP0202OpsMag1.tyMsgBoxUnloadAsk);

			IF tyP0202OpsMag1.tyMsgBoxUnloadAsk.tyBtnYes.bRtCompl = TRUE THEN
				tyP0202OpsMag1.tyMsgBoxUnloadAsk.tyBtnYes.bRtCompl	:= FALSE;
				tyP0202OpsMag1.tyMsgBoxUnloadAsk.tyBtnYes.bValue	:= FALSE;

				p_tyC0008MsgBox ACCESS ADR(tyP0202OpsMag1.tyMsgBoxHide);

				bUnloadMag	:= TRUE;

				tyP0202OpsMag1.tyOps.tyBtnUnloadMag.bRtCompl	:= FALSE;

			ELSIF tyP0202OpsMag1.tyMsgBoxUnloadAsk.tyBtnNo.bRtCompl = TRUE THEN
				tyP0202OpsMag1.tyMsgBoxUnloadAsk.tyBtnNo.bRtCompl	:= FALSE;
				tyP0202OpsMag1.tyMsgBoxUnloadAsk.tyBtnNo.bValue		:= FALSE;

				p_tyC0008MsgBox ACCESS ADR(tyP0202OpsMag1.tyMsgBoxHide);

				tyP0202OpsMag1.tyOps.tyBtnUnloadMag.bRtCompl	:= FALSE;

			END_IF

		ELSE

			p_tyC0008MsgBox ACCESS ADR(tyP0202OpsMag1.tyMsgBoxResumeAsk);

			IF tyP0202OpsMag1.tyMsgBoxResumeAsk.tyBtnYes.bRtCompl = TRUE THEN
				tyP0202OpsMag1.tyMsgBoxResumeAsk.tyBtnYes.bRtCompl	:= FALSE;
				tyP0202OpsMag1.tyMsgBoxResumeAsk.tyBtnYes.bValue	:= FALSE;

				p_tyC0008MsgBox ACCESS ADR(tyP0202OpsMag1.tyMsgBoxHide);

				bUnloadMag	:= FALSE;

				tyP0202OpsMag1.tyOps.tyBtnUnloadMag.bRtCompl	:= FALSE;

			ELSIF tyP0202OpsMag1.tyMsgBoxResumeAsk.tyBtnNo.bRtCompl = TRUE THEN
				tyP0202OpsMag1.tyMsgBoxResumeAsk.tyBtnNo.bRtCompl	:= FALSE;
				tyP0202OpsMag1.tyMsgBoxResumeAsk.tyBtnNo.bValue		:= FALSE;

				p_tyC0008MsgBox ACCESS ADR(tyP0202OpsMag1.tyMsgBoxHide);

				tyP0202OpsMag1.tyOps.tyBtnUnloadMag.bRtCompl	:= FALSE;

			END_IF

		END_IF

	ELSIF tyP0203OpsMag2.tyOps.tyBtnUnloadMag.bRtCompl = TRUE THEN

		IF bUnloadMag = FALSE THEN

			p_tyC0008MsgBox ACCESS ADR(tyP0203OpsMag2.tyMsgBoxUnloadAsk);

			IF tyP0203OpsMag2.tyMsgBoxUnloadAsk.tyBtnYes.bRtCompl = TRUE THEN
				tyP0203OpsMag2.tyMsgBoxUnloadAsk.tyBtnYes.bRtCompl	:= FALSE;
				tyP0203OpsMag2.tyMsgBoxUnloadAsk.tyBtnYes.bValue	:= FALSE;

				p_tyC0008MsgBox ACCESS ADR(tyP0203OpsMag2.tyMsgBoxHide);

				bUnloadMag	:= TRUE;

				tyP0203OpsMag2.tyOps.tyBtnUnloadMag.bRtCompl	:= FALSE;

			ELSIF tyP0203OpsMag2.tyMsgBoxUnloadAsk.tyBtnNo.bRtCompl = TRUE THEN
				tyP0203OpsMag2.tyMsgBoxUnloadAsk.tyBtnNo.bRtCompl	:= FALSE;
				tyP0203OpsMag2.tyMsgBoxUnloadAsk.tyBtnNo.bValue		:= FALSE;

				p_tyC0008MsgBox ACCESS ADR(tyP0203OpsMag2.tyMsgBoxHide);

				tyP0203OpsMag2.tyOps.tyBtnUnloadMag.bRtCompl	:= FALSE;

			END_IF

		ELSE

			p_tyC0008MsgBox ACCESS ADR(tyP0203OpsMag2.tyMsgBoxResumeAsk);

			IF tyP0203OpsMag2.tyMsgBoxResumeAsk.tyBtnYes.bRtCompl = TRUE THEN
				tyP0203OpsMag2.tyMsgBoxResumeAsk.tyBtnYes.bRtCompl	:= FALSE;
				tyP0203OpsMag2.tyMsgBoxResumeAsk.tyBtnYes.bValue	:= FALSE;

				p_tyC0008MsgBox ACCESS ADR(tyP0203OpsMag2.tyMsgBoxHide);

				bUnloadMag	:= FALSE;

				tyP0203OpsMag2.tyOps.tyBtnUnloadMag.bRtCompl	:= FALSE;

			ELSIF tyP0203OpsMag2.tyMsgBoxResumeAsk.tyBtnNo.bRtCompl = TRUE THEN
				tyP0203OpsMag2.tyMsgBoxResumeAsk.tyBtnNo.bRtCompl	:= FALSE;
				tyP0203OpsMag2.tyMsgBoxResumeAsk.tyBtnNo.bValue		:= FALSE;

				p_tyC0008MsgBox ACCESS ADR(tyP0203OpsMag2.tyMsgBoxHide);

				tyP0203OpsMag2.tyOps.tyBtnUnloadMag.bRtCompl	:= FALSE;

			END_IF

		END_IF

	ELSIF tyP0204OpsMag3.tyOps.tyBtnUnloadMag.bRtCompl = TRUE THEN

		IF bUnloadMag = FALSE THEN

			p_tyC0008MsgBox ACCESS ADR(tyP0204OpsMag3.tyMsgBoxUnloadAsk);

			IF tyP0204OpsMag3.tyMsgBoxUnloadAsk.tyBtnYes.bRtCompl = TRUE THEN
				tyP0204OpsMag3.tyMsgBoxUnloadAsk.tyBtnYes.bRtCompl	:= FALSE;
				tyP0204OpsMag3.tyMsgBoxUnloadAsk.tyBtnYes.bValue	:= FALSE;

				p_tyC0008MsgBox ACCESS ADR(tyP0204OpsMag3.tyMsgBoxHide);

				bUnloadMag	:= TRUE;

				tyP0204OpsMag3.tyOps.tyBtnUnloadMag.bRtCompl	:= FALSE;

			ELSIF tyP0204OpsMag3.tyMsgBoxUnloadAsk.tyBtnNo.bRtCompl = TRUE THEN
				tyP0204OpsMag3.tyMsgBoxUnloadAsk.tyBtnNo.bRtCompl	:= FALSE;
				tyP0204OpsMag3.tyMsgBoxUnloadAsk.tyBtnNo.bValue		:= FALSE;

				p_tyC0008MsgBox ACCESS ADR(tyP0204OpsMag3.tyMsgBoxHide);

				tyP0204OpsMag3.tyOps.tyBtnUnloadMag.bRtCompl	:= FALSE;

			END_IF

		ELSE

			p_tyC0008MsgBox ACCESS ADR(tyP0204OpsMag3.tyMsgBoxResumeAsk);

			IF tyP0204OpsMag3.tyMsgBoxResumeAsk.tyBtnYes.bRtCompl = TRUE THEN
				tyP0204OpsMag3.tyMsgBoxResumeAsk.tyBtnYes.bRtCompl	:= FALSE;
				tyP0204OpsMag3.tyMsgBoxResumeAsk.tyBtnYes.bValue	:= FALSE;

				p_tyC0008MsgBox ACCESS ADR(tyP0204OpsMag3.tyMsgBoxHide);

				bUnloadMag	:= FALSE;

				tyP0204OpsMag3.tyOps.tyBtnUnloadMag.bRtCompl	:= FALSE;

			ELSIF tyP0204OpsMag3.tyMsgBoxResumeAsk.tyBtnNo.bRtCompl = TRUE THEN
				tyP0204OpsMag3.tyMsgBoxResumeAsk.tyBtnNo.bRtCompl	:= FALSE;
				tyP0204OpsMag3.tyMsgBoxResumeAsk.tyBtnNo.bValue		:= FALSE;

				p_tyC0008MsgBox ACCESS ADR(tyP0204OpsMag3.tyMsgBoxHide);

				tyP0204OpsMag3.tyOps.tyBtnUnloadMag.bRtCompl	:= FALSE;

			END_IF

		END_IF

	ELSIF tyP0206OpsMag4.tyOps.tyBtnUnloadMag.bRtCompl = TRUE THEN

		IF bUnloadMag = FALSE THEN

			p_tyC0008MsgBox ACCESS ADR(tyP0206OpsMag4.tyMsgBoxUnloadAsk);

			IF tyP0206OpsMag4.tyMsgBoxUnloadAsk.tyBtnYes.bRtCompl = TRUE THEN
				tyP0206OpsMag4.tyMsgBoxUnloadAsk.tyBtnYes.bRtCompl	:= FALSE;
				tyP0206OpsMag4.tyMsgBoxUnloadAsk.tyBtnYes.bValue	:= FALSE;

				p_tyC0008MsgBox ACCESS ADR(tyP0206OpsMag4.tyMsgBoxHide);

				bUnloadMag	:= TRUE;

				tyP0206OpsMag4.tyOps.tyBtnUnloadMag.bRtCompl	:= FALSE;

			ELSIF tyP0206OpsMag4.tyMsgBoxUnloadAsk.tyBtnNo.bRtCompl = TRUE THEN
				tyP0206OpsMag4.tyMsgBoxUnloadAsk.tyBtnNo.bRtCompl	:= FALSE;
				tyP0206OpsMag4.tyMsgBoxUnloadAsk.tyBtnNo.bValue		:= FALSE;

				p_tyC0008MsgBox ACCESS ADR(tyP0206OpsMag4.tyMsgBoxHide);

				tyP0206OpsMag4.tyOps.tyBtnUnloadMag.bRtCompl	:= FALSE;

			END_IF

		ELSE

			p_tyC0008MsgBox ACCESS ADR(tyP0206OpsMag4.tyMsgBoxResumeAsk);

			IF tyP0206OpsMag4.tyMsgBoxResumeAsk.tyBtnYes.bRtCompl = TRUE THEN
				tyP0206OpsMag4.tyMsgBoxResumeAsk.tyBtnYes.bRtCompl	:= FALSE;
				tyP0206OpsMag4.tyMsgBoxResumeAsk.tyBtnYes.bValue	:= FALSE;

				p_tyC0008MsgBox ACCESS ADR(tyP0206OpsMag4.tyMsgBoxHide);

				bUnloadMag	:= FALSE;

				tyP0206OpsMag4.tyOps.tyBtnUnloadMag.bRtCompl	:= FALSE;

			ELSIF tyP0206OpsMag4.tyMsgBoxResumeAsk.tyBtnNo.bRtCompl = TRUE THEN
				tyP0206OpsMag4.tyMsgBoxResumeAsk.tyBtnNo.bRtCompl	:= FALSE;
				tyP0206OpsMag4.tyMsgBoxResumeAsk.tyBtnNo.bValue		:= FALSE;

				p_tyC0008MsgBox ACCESS ADR(tyP0206OpsMag4.tyMsgBoxHide);

				tyP0206OpsMag4.tyOps.tyBtnUnloadMag.bRtCompl	:= FALSE;

			END_IF

		END_IF
	END_IF

	//Display
	tyP0202OpsMag1.tyOps.tyBtnUnloadMag.bRtLk	:= p_bOpsStatusStop = FALSE AND bUnloadMag AND NOT p_bOpsLifMagLDUnloading;
	tyP0203OpsMag2.tyOps.tyBtnUnloadMag.bRtLk	:= p_bOpsStatusStop = FALSE AND bUnloadMag AND NOT p_bOpsLifMagLDUnloading;
	tyP0204OpsMag3.tyOps.tyBtnUnloadMag.bRtLk	:= p_bOpsStatusStop = FALSE AND bUnloadMag AND NOT p_bOpsLifMagLDUnloading;
	tyP0206OpsMag4.tyOps.tyBtnUnloadMag.bRtLk	:= p_bOpsStatusStop = FALSE AND bUnloadMag AND NOT p_bOpsLifMagLDUnloading;

	IF p_bOpsStatusStop = FALSE AND p_bOpsLifMagLDUnloading = TRUE THEN
		tyP0202OpsMag1.tyOps.tyBtnUnloadMag.usiTxtIdx	:= 1;
		tyP0203OpsMag2.tyOps.tyBtnUnloadMag.usiTxtIdx	:= 1;
		tyP0204OpsMag3.tyOps.tyBtnUnloadMag.usiTxtIdx	:= 1;
		tyP0206OpsMag4.tyOps.tyBtnUnloadMag.usiTxtIdx	:= 1;
	ELSE
		tyP0202OpsMag1.tyOps.tyBtnUnloadMag.usiTxtIdx	:= 0;
		tyP0203OpsMag2.tyOps.tyBtnUnloadMag.usiTxtIdx	:= 0;
		tyP0204OpsMag3.tyOps.tyBtnUnloadMag.usiTxtIdx	:= 0;
		tyP0206OpsMag4.tyOps.tyBtnUnloadMag.usiTxtIdx	:= 0;
	END_IF

	IF p_bOpsStatusStop = FALSE AND bUnloadMag = TRUE AND p_bOpsLifMagLDUnloading = TRUE THEN

		fbUnloadBlinkTm(IN := TRUE);

		IF fbUnloadBlinkTm.Q = TRUE THEN
			fbUnloadBlinkTm(IN := FALSE);

			IF tyP0202OpsMag1.tyOps.tyBitmapUnloadMag.usiValueIdx = 0 THEN
				tyP0202OpsMag1.tyOps.tyBitmapUnloadMag.usiValueIdx	:= 3;
				tyP0203OpsMag2.tyOps.tyBitmapUnloadMag.usiValueIdx	:= 3;
				tyP0204OpsMag3.tyOps.tyBitmapUnloadMag.usiValueIdx	:= 3;
				tyP0206OpsMag4.tyOps.tyBitmapUnloadMag.usiValueIdx	:= 3;
			ELSE
				tyP0202OpsMag1.tyOps.tyBitmapUnloadMag.usiValueIdx	:= 0;
				tyP0203OpsMag2.tyOps.tyBitmapUnloadMag.usiValueIdx	:= 0;
				tyP0204OpsMag3.tyOps.tyBitmapUnloadMag.usiValueIdx	:= 0;
				tyP0206OpsMag4.tyOps.tyBitmapUnloadMag.usiValueIdx	:= 0;
			END_IF

		END_IF

	ELSIF p_bOpsStatusStop = FALSE AND bUnloadMag = TRUE THEN

		fbUnloadBlinkTm(IN := FALSE);

		tyP0202OpsMag1.tyOps.tyBitmapUnloadMag.usiValueIdx	:= 1;
		tyP0203OpsMag2.tyOps.tyBitmapUnloadMag.usiValueIdx	:= 1;
		tyP0204OpsMag3.tyOps.tyBitmapUnloadMag.usiValueIdx	:= 1;
		tyP0206OpsMag4.tyOps.tyBitmapUnloadMag.usiValueIdx	:= 1;
	ELSE

		fbUnloadBlinkTm(IN := FALSE);

		tyP0202OpsMag1.tyOps.tyBitmapUnloadMag.usiValueIdx	:= 0;
		tyP0203OpsMag2.tyOps.tyBitmapUnloadMag.usiValueIdx	:= 0;
		tyP0204OpsMag3.tyOps.tyBitmapUnloadMag.usiValueIdx	:= 0;
		tyP0206OpsMag4.tyOps.tyBitmapUnloadMag.usiValueIdx	:= 0;
	END_IF

	//Mask
	tyP0202OpsMag1.tyOps.tyBtnUnloadMag.uiMaskRtStat.0	:= NOT p_bOpsStatusStop;
	tyP0203OpsMag2.tyOps.tyBtnUnloadMag.uiMaskRtStat.0	:= NOT p_bOpsStatusStop;
	tyP0204OpsMag3.tyOps.tyBtnUnloadMag.uiMaskRtStat.0	:= NOT p_bOpsStatusStop;
	tyP0206OpsMag4.tyOps.tyBtnUnloadMag.uiMaskRtStat.0	:= NOT p_bOpsStatusStop;

END_ACTION
```

#### Act_OptP0202ToP0204_P0003UnloadMag.st - not listed in the package file held
```iecst
ACTION Act_OptP0202ToP0204_P0003UnloadMag:

	//Reset
	IF EDGEPOS(p_bOpsStatusStop) THEN
		bUnloadMag	:= FALSE;

		tyP0202OpsMag1.tyOps.tyBtnUnloadMag.bRtCompl	:= FALSE;
		tyP0203OpsMag2.tyOps.tyBtnUnloadMag.bRtCompl	:= FALSE;
		tyP0204OpsMag3.tyOps.tyBtnUnloadMag.bRtCompl	:= FALSE;
		tyP0003MMenu.tyMMenuBtn.tyBtnUnload.bRtCompl := FALSE;

		p_tyC0008MsgBox ACCESS ADR(tyP0202OpsMag1.tyMsgBoxHide);
		p_tyC0008MsgBox ACCESS ADR(tyP0203OpsMag2.tyMsgBoxHide);
		p_tyC0008MsgBox ACCESS ADR(tyP0204OpsMag3.tyMsgBoxHide);
	END_IF

	//Control
	IF tyP0202OpsMag1.tyOps.tyBtnUnloadMag.bRtCompl = TRUE THEN

		IF bUnloadMag = FALSE THEN

			p_tyC0008MsgBox ACCESS ADR(tyP0202OpsMag1.tyMsgBoxUnloadAsk);

			IF tyP0202OpsMag1.tyMsgBoxUnloadAsk.tyBtnYes.bRtCompl = TRUE THEN
				tyP0202OpsMag1.tyMsgBoxUnloadAsk.tyBtnYes.bRtCompl	:= FALSE;
				tyP0202OpsMag1.tyMsgBoxUnloadAsk.tyBtnYes.bValue	:= FALSE;

				p_tyC0008MsgBox ACCESS ADR(tyP0202OpsMag1.tyMsgBoxHide);

				bUnloadMag	:= TRUE;

				tyP0202OpsMag1.tyOps.tyBtnUnloadMag.bRtCompl	:= FALSE;

			ELSIF tyP0202OpsMag1.tyMsgBoxUnloadAsk.tyBtnNo.bRtCompl = TRUE THEN
				tyP0202OpsMag1.tyMsgBoxUnloadAsk.tyBtnNo.bRtCompl	:= FALSE;
				tyP0202OpsMag1.tyMsgBoxUnloadAsk.tyBtnNo.bValue		:= FALSE;

				p_tyC0008MsgBox ACCESS ADR(tyP0202OpsMag1.tyMsgBoxHide);

				tyP0202OpsMag1.tyOps.tyBtnUnloadMag.bRtCompl	:= FALSE;

			END_IF

		ELSE

			p_tyC0008MsgBox ACCESS ADR(tyP0202OpsMag1.tyMsgBoxResumeAsk);

			IF tyP0202OpsMag1.tyMsgBoxResumeAsk.tyBtnYes.bRtCompl = TRUE THEN
				tyP0202OpsMag1.tyMsgBoxResumeAsk.tyBtnYes.bRtCompl	:= FALSE;
				tyP0202OpsMag1.tyMsgBoxResumeAsk.tyBtnYes.bValue	:= FALSE;

				p_tyC0008MsgBox ACCESS ADR(tyP0202OpsMag1.tyMsgBoxHide);

				bUnloadMag	:= FALSE;

				tyP0202OpsMag1.tyOps.tyBtnUnloadMag.bRtCompl	:= FALSE;

			ELSIF tyP0202OpsMag1.tyMsgBoxResumeAsk.tyBtnNo.bRtCompl = TRUE THEN
				tyP0202OpsMag1.tyMsgBoxResumeAsk.tyBtnNo.bRtCompl	:= FALSE;
				tyP0202OpsMag1.tyMsgBoxResumeAsk.tyBtnNo.bValue		:= FALSE;

				p_tyC0008MsgBox ACCESS ADR(tyP0202OpsMag1.tyMsgBoxHide);

				tyP0202OpsMag1.tyOps.tyBtnUnloadMag.bRtCompl	:= FALSE;

			END_IF

		END_IF

	ELSIF tyP0203OpsMag2.tyOps.tyBtnUnloadMag.bRtCompl = TRUE THEN

		IF bUnloadMag = FALSE THEN

			p_tyC0008MsgBox ACCESS ADR(tyP0203OpsMag2.tyMsgBoxUnloadAsk);

			IF tyP0203OpsMag2.tyMsgBoxUnloadAsk.tyBtnYes.bRtCompl = TRUE THEN
				tyP0203OpsMag2.tyMsgBoxUnloadAsk.tyBtnYes.bRtCompl	:= FALSE;
				tyP0203OpsMag2.tyMsgBoxUnloadAsk.tyBtnYes.bValue	:= FALSE;

				p_tyC0008MsgBox ACCESS ADR(tyP0203OpsMag2.tyMsgBoxHide);

				bUnloadMag	:= TRUE;

				tyP0203OpsMag2.tyOps.tyBtnUnloadMag.bRtCompl	:= FALSE;

			ELSIF tyP0203OpsMag2.tyMsgBoxUnloadAsk.tyBtnNo.bRtCompl = TRUE THEN
				tyP0203OpsMag2.tyMsgBoxUnloadAsk.tyBtnNo.bRtCompl	:= FALSE;
				tyP0203OpsMag2.tyMsgBoxUnloadAsk.tyBtnNo.bValue		:= FALSE;

				p_tyC0008MsgBox ACCESS ADR(tyP0203OpsMag2.tyMsgBoxHide);

				tyP0203OpsMag2.tyOps.tyBtnUnloadMag.bRtCompl	:= FALSE;

			END_IF

		ELSE

			p_tyC0008MsgBox ACCESS ADR(tyP0203OpsMag2.tyMsgBoxResumeAsk);

			IF tyP0203OpsMag2.tyMsgBoxResumeAsk.tyBtnYes.bRtCompl = TRUE THEN
				tyP0203OpsMag2.tyMsgBoxResumeAsk.tyBtnYes.bRtCompl	:= FALSE;
				tyP0203OpsMag2.tyMsgBoxResumeAsk.tyBtnYes.bValue	:= FALSE;

				p_tyC0008MsgBox ACCESS ADR(tyP0203OpsMag2.tyMsgBoxHide);

				bUnloadMag	:= FALSE;

				tyP0203OpsMag2.tyOps.tyBtnUnloadMag.bRtCompl	:= FALSE;

			ELSIF tyP0203OpsMag2.tyMsgBoxResumeAsk.tyBtnNo.bRtCompl = TRUE THEN
				tyP0203OpsMag2.tyMsgBoxResumeAsk.tyBtnNo.bRtCompl	:= FALSE;
				tyP0203OpsMag2.tyMsgBoxResumeAsk.tyBtnNo.bValue		:= FALSE;

				p_tyC0008MsgBox ACCESS ADR(tyP0203OpsMag2.tyMsgBoxHide);

				tyP0203OpsMag2.tyOps.tyBtnUnloadMag.bRtCompl	:= FALSE;

			END_IF

		END_IF

	ELSIF tyP0204OpsMag3.tyOps.tyBtnUnloadMag.bRtCompl = TRUE THEN

		IF bUnloadMag = FALSE THEN

			p_tyC0008MsgBox ACCESS ADR(tyP0204OpsMag3.tyMsgBoxUnloadAsk);

			IF tyP0204OpsMag3.tyMsgBoxUnloadAsk.tyBtnYes.bRtCompl = TRUE THEN
				tyP0204OpsMag3.tyMsgBoxUnloadAsk.tyBtnYes.bRtCompl	:= FALSE;
				tyP0204OpsMag3.tyMsgBoxUnloadAsk.tyBtnYes.bValue	:= FALSE;

				p_tyC0008MsgBox ACCESS ADR(tyP0204OpsMag3.tyMsgBoxHide);

				bUnloadMag	:= TRUE;

				tyP0204OpsMag3.tyOps.tyBtnUnloadMag.bRtCompl	:= FALSE;

			ELSIF tyP0204OpsMag3.tyMsgBoxUnloadAsk.tyBtnNo.bRtCompl = TRUE THEN
				tyP0204OpsMag3.tyMsgBoxUnloadAsk.tyBtnNo.bRtCompl	:= FALSE;
				tyP0204OpsMag3.tyMsgBoxUnloadAsk.tyBtnNo.bValue		:= FALSE;

				p_tyC0008MsgBox ACCESS ADR(tyP0204OpsMag3.tyMsgBoxHide);

				tyP0204OpsMag3.tyOps.tyBtnUnloadMag.bRtCompl	:= FALSE;

			END_IF

		ELSE

			p_tyC0008MsgBox ACCESS ADR(tyP0204OpsMag3.tyMsgBoxResumeAsk);

			IF tyP0204OpsMag3.tyMsgBoxResumeAsk.tyBtnYes.bRtCompl = TRUE THEN
				tyP0204OpsMag3.tyMsgBoxResumeAsk.tyBtnYes.bRtCompl	:= FALSE;
				tyP0204OpsMag3.tyMsgBoxResumeAsk.tyBtnYes.bValue	:= FALSE;

				p_tyC0008MsgBox ACCESS ADR(tyP0204OpsMag3.tyMsgBoxHide);

				bUnloadMag	:= FALSE;

				tyP0204OpsMag3.tyOps.tyBtnUnloadMag.bRtCompl	:= FALSE;

			ELSIF tyP0204OpsMag3.tyMsgBoxResumeAsk.tyBtnNo.bRtCompl = TRUE THEN
				tyP0204OpsMag3.tyMsgBoxResumeAsk.tyBtnNo.bRtCompl	:= FALSE;
				tyP0204OpsMag3.tyMsgBoxResumeAsk.tyBtnNo.bValue		:= FALSE;

				p_tyC0008MsgBox ACCESS ADR(tyP0204OpsMag3.tyMsgBoxHide);

				tyP0204OpsMag3.tyOps.tyBtnUnloadMag.bRtCompl	:= FALSE;

			END_IF

		END_IF

	ELSIF tyP0206OpsMag4.tyOps.tyBtnUnloadMag.bRtCompl = TRUE THEN

		IF bUnloadMag = FALSE THEN

			p_tyC0008MsgBox ACCESS ADR(tyP0206OpsMag4.tyMsgBoxUnloadAsk);

			IF tyP0206OpsMag4.tyMsgBoxUnloadAsk.tyBtnYes.bRtCompl = TRUE THEN
				tyP0206OpsMag4.tyMsgBoxUnloadAsk.tyBtnYes.bRtCompl	:= FALSE;
				tyP0206OpsMag4.tyMsgBoxUnloadAsk.tyBtnYes.bValue	:= FALSE;

				p_tyC0008MsgBox ACCESS ADR(tyP0206OpsMag4.tyMsgBoxHide);

				bUnloadMag	:= TRUE;

				tyP0206OpsMag4.tyOps.tyBtnUnloadMag.bRtCompl	:= FALSE;

			ELSIF tyP0206OpsMag4.tyMsgBoxUnloadAsk.tyBtnNo.bRtCompl = TRUE THEN
				tyP0206OpsMag4.tyMsgBoxUnloadAsk.tyBtnNo.bRtCompl	:= FALSE;
				tyP0206OpsMag4.tyMsgBoxUnloadAsk.tyBtnNo.bValue		:= FALSE;

				p_tyC0008MsgBox ACCESS ADR(tyP0206OpsMag4.tyMsgBoxHide);

				tyP0206OpsMag4.tyOps.tyBtnUnloadMag.bRtCompl	:= FALSE;

			END_IF

		ELSE

			p_tyC0008MsgBox ACCESS ADR(tyP0206OpsMag4.tyMsgBoxResumeAsk);

			IF tyP0206OpsMag4.tyMsgBoxResumeAsk.tyBtnYes.bRtCompl = TRUE THEN
				tyP0206OpsMag4.tyMsgBoxResumeAsk.tyBtnYes.bRtCompl	:= FALSE;
				tyP0206OpsMag4.tyMsgBoxResumeAsk.tyBtnYes.bValue	:= FALSE;

				p_tyC0008MsgBox ACCESS ADR(tyP0206OpsMag4.tyMsgBoxHide);

				bUnloadMag	:= FALSE;

				tyP0206OpsMag4.tyOps.tyBtnUnloadMag.bRtCompl	:= FALSE;

			ELSIF tyP0206OpsMag4.tyMsgBoxResumeAsk.tyBtnNo.bRtCompl = TRUE THEN
				tyP0206OpsMag4.tyMsgBoxResumeAsk.tyBtnNo.bRtCompl	:= FALSE;
				tyP0206OpsMag4.tyMsgBoxResumeAsk.tyBtnNo.bValue		:= FALSE;

				p_tyC0008MsgBox ACCESS ADR(tyP0206OpsMag4.tyMsgBoxHide);

				tyP0206OpsMag4.tyOps.tyBtnUnloadMag.bRtCompl	:= FALSE;

			END_IF

		END_IF
	ELSIF tyP0003MMenu.tyMMenuBtn.tyBtnUnload.bRtCompl = TRUE THEN

		IF bUnloadMag = FALSE THEN

			p_tyC0008MsgBox ACCESS ADR(tyP0003MMenu.tyMsgBoxUnloadAsk);

			IF tyP0003MMenu.tyMsgBoxUnloadAsk.tyBtnYes.bRtCompl = TRUE THEN
				tyP0003MMenu.tyMsgBoxUnloadAsk.tyBtnYes.bRtCompl	:= FALSE;
				tyP0003MMenu.tyMsgBoxUnloadAsk.tyBtnYes.bValue	:= FALSE;

				p_tyC0008MsgBox ACCESS ADR(tyP0003MMenu.tyMsgBoxHide);

				bUnloadMag	:= TRUE;

				tyP0003MMenu.tyMMenuBtn.tyBtnUnload.bRtCompl	:= FALSE;

			ELSIF tyP0003MMenu.tyMsgBoxUnloadAsk.tyBtnNo.bRtCompl = TRUE THEN
				tyP0003MMenu.tyMsgBoxUnloadAsk.tyBtnNo.bRtCompl	:= FALSE;
				tyP0003MMenu.tyMsgBoxUnloadAsk.tyBtnNo.bValue	:= FALSE;

				p_tyC0008MsgBox ACCESS ADR(tyP0003MMenu.tyMsgBoxHide);

				tyP0003MMenu.tyMMenuBtn.tyBtnUnload.bRtCompl	:= FALSE;

			END_IF

		ELSE

			p_tyC0008MsgBox ACCESS ADR(tyP0003MMenu.tyMsgBoxResumeAsk);

			IF tyP0003MMenu.tyMsgBoxResumeAsk.tyBtnYes.bRtCompl = TRUE THEN
				tyP0003MMenu.tyMsgBoxResumeAsk.tyBtnYes.bRtCompl	:= FALSE;
				tyP0003MMenu.tyMsgBoxResumeAsk.tyBtnYes.bValue	:= FALSE;

				p_tyC0008MsgBox ACCESS ADR(tyP0003MMenu.tyMsgBoxHide);

				bUnloadMag	:= FALSE;

				tyP0003MMenu.tyMMenuBtn.tyBtnUnload.bRtCompl	:= FALSE;

			ELSIF tyP0003MMenu.tyMsgBoxResumeAsk.tyBtnNo.bRtCompl = TRUE THEN
				tyP0003MMenu.tyMsgBoxResumeAsk.tyBtnNo.bRtCompl	:= FALSE;
				tyP0003MMenu.tyMsgBoxResumeAsk.tyBtnNo.bValue		:= FALSE;

				p_tyC0008MsgBox ACCESS ADR(tyP0003MMenu.tyMsgBoxHide);

				tyP0003MMenu.tyMMenuBtn.tyBtnUnload.bRtCompl	:= FALSE;

			END_IF

		END_IF

	END_IF

	//Display
	tyP0202OpsMag1.tyOps.tyBtnUnloadMag.bRtLk	:= p_bOpsStatusStop = FALSE AND bUnloadMag AND NOT p_bOpsLifMagLDUnloading;
	tyP0203OpsMag2.tyOps.tyBtnUnloadMag.bRtLk	:= p_bOpsStatusStop = FALSE AND bUnloadMag AND NOT p_bOpsLifMagLDUnloading;
	tyP0204OpsMag3.tyOps.tyBtnUnloadMag.bRtLk	:= p_bOpsStatusStop = FALSE AND bUnloadMag AND NOT p_bOpsLifMagLDUnloading;
	tyP0206OpsMag4.tyOps.tyBtnUnloadMag.bRtLk	:= p_bOpsStatusStop = FALSE AND bUnloadMag AND NOT p_bOpsLifMagLDUnloading;
	tyP0003MMenu.tyMMenuBtn.tyBtnUnload.bRtLk 	:= p_bOpsStatusStop = FALSE AND bUnloadMag AND NOT p_bOpsLifMagLDUnloading;

	IF p_bOpsStatusStop = FALSE AND p_bOpsLifMagLDUnloading = TRUE THEN
		tyP0202OpsMag1.tyOps.tyBtnUnloadMag.usiTxtIdx	:= 1;
		tyP0203OpsMag2.tyOps.tyBtnUnloadMag.usiTxtIdx	:= 1;
		tyP0204OpsMag3.tyOps.tyBtnUnloadMag.usiTxtIdx	:= 1;
		tyP0206OpsMag4.tyOps.tyBtnUnloadMag.usiTxtIdx	:= 1;

		tyP0003MMenu.tyMMenuBtn.tyBtnUnload.usiTxtIdx	:= 30; //Text group - Main Menu
	ELSE
		tyP0202OpsMag1.tyOps.tyBtnUnloadMag.usiTxtIdx	:= 0;
		tyP0203OpsMag2.tyOps.tyBtnUnloadMag.usiTxtIdx	:= 0;
		tyP0204OpsMag3.tyOps.tyBtnUnloadMag.usiTxtIdx	:= 0;
		tyP0206OpsMag4.tyOps.tyBtnUnloadMag.usiTxtIdx	:= 0;

		tyP0003MMenu.tyMMenuBtn.tyBtnUnload.usiTxtIdx	:= 5; //Text group - Main Menu
	END_IF

	IF p_bOpsStatusStop = FALSE AND bUnloadMag = TRUE AND p_bOpsLifMagLDUnloading = TRUE THEN

		fbUnloadBlinkTm(IN := TRUE);

		IF fbUnloadBlinkTm.Q = TRUE THEN
			fbUnloadBlinkTm(IN := FALSE);

			IF tyP0202OpsMag1.tyOps.tyBitmapUnloadMag.usiValueIdx = 0 THEN
				tyP0202OpsMag1.tyOps.tyBitmapUnloadMag.usiValueIdx	:= 3;
				tyP0203OpsMag2.tyOps.tyBitmapUnloadMag.usiValueIdx	:= 3;
				tyP0204OpsMag3.tyOps.tyBitmapUnloadMag.usiValueIdx	:= 3;
				tyP0206OpsMag4.tyOps.tyBitmapUnloadMag.usiValueIdx	:= 3;

				tyP0003MMenu.tyMMenuBtn.tyBtnUnload.usiBitmapIdx    := 4; //Yellow
			ELSE
				tyP0202OpsMag1.tyOps.tyBitmapUnloadMag.usiValueIdx	:= 0;
				tyP0203OpsMag2.tyOps.tyBitmapUnloadMag.usiValueIdx	:= 0;
				tyP0204OpsMag3.tyOps.tyBitmapUnloadMag.usiValueIdx	:= 0;
				tyP0206OpsMag4.tyOps.tyBitmapUnloadMag.usiValueIdx	:= 0;

				tyP0003MMenu.tyMMenuBtn.tyBtnUnload.usiBitmapIdx    := 0; //Silver
			END_IF

		END_IF

	ELSIF p_bOpsStatusStop = FALSE AND bUnloadMag = TRUE THEN

		fbUnloadBlinkTm(IN := FALSE);

		tyP0202OpsMag1.tyOps.tyBitmapUnloadMag.usiValueIdx	:= 1;
		tyP0203OpsMag2.tyOps.tyBitmapUnloadMag.usiValueIdx	:= 1;
		tyP0204OpsMag3.tyOps.tyBitmapUnloadMag.usiValueIdx	:= 1;
		tyP0206OpsMag4.tyOps.tyBitmapUnloadMag.usiValueIdx	:= 1;

		tyP0003MMenu.tyMMenuBtn.tyBtnUnload.usiBitmapIdx    := 1; //Green
	ELSE

		fbUnloadBlinkTm(IN := FALSE);

		tyP0202OpsMag1.tyOps.tyBitmapUnloadMag.usiValueIdx	:= 0;
		tyP0203OpsMag2.tyOps.tyBitmapUnloadMag.usiValueIdx	:= 0;
		tyP0204OpsMag3.tyOps.tyBitmapUnloadMag.usiValueIdx	:= 0;
		tyP0206OpsMag4.tyOps.tyBitmapUnloadMag.usiValueIdx	:= 0;
	END_IF

	//Mask
	tyP0202OpsMag1.tyOps.tyBtnUnloadMag.uiMaskRtStat.0	:= NOT p_bOpsStatusStop;
	tyP0203OpsMag2.tyOps.tyBtnUnloadMag.uiMaskRtStat.0	:= NOT p_bOpsStatusStop;
	tyP0204OpsMag3.tyOps.tyBtnUnloadMag.uiMaskRtStat.0	:= NOT p_bOpsStatusStop;
	tyP0206OpsMag4.tyOps.tyBtnUnloadMag.uiMaskRtStat.0	:= NOT p_bOpsStatusStop;

	tyP0003MMenu.tyMMenuBtn.tyBtnUnload.uiMaskRtStat.0 := NOT p_bOpsStatusStop;

END_ACTION
```

#### Act_EntP0205Disp.st
```iecst
ACTION Act_EntP0205Disp:

	//Access Address
	p_tyC0004Navi ACCESS ADR(tyP0205OpsAIV.tyNaviBack);

	p_tyC0005Main ACCESS ADR(tyCommon.tyMain);

	p_tyC0007Notif ACCESS ADR(tyCommon.tyNotif);

	p_tyC0008MsgBox ACCESS ADR(tyP0205OpsAIV.tyMsgBoxHide);

	p_tyC0009Info ACCESS ADR(tyCommon.tyInfo);

	p_tyP0205IOMonitor ACCESS ADR(tyP0205OpsAIV.tyIOMonitor);

	tyP0205OpsAIV.tyIOMonitor.tyBitmapAIVSLarge1.uiRtStat.0 := p_tyMcParamCurr.bAIVSizeDisabled;
	tyP0205OpsAIV.tyIOMonitor.tyBitmapAIVSLarge2.uiRtStat.0 := p_tyMcParamCurr.bAIVSizeDisabled;
	tyP0205OpsAIV.tyIOMonitor.tyBitmapAIVSLarge3.uiRtStat.0 := p_tyMcParamCurr.bAIVSizeDisabled;
	tyP0205OpsAIV.tyIOMonitor.tyBitmapAIVSLarge4.uiRtStat.0 := p_tyMcParamCurr.bAIVSizeDisabled;

	tyP0205OpsAIV.tyIOMonitor.tyBitmapMagSLarge1.uiRtStat.0 := p_tyMcParamCurr.bAIVSizeDisabled;
	tyP0205OpsAIV.tyIOMonitor.tyBitmapMagSLarge2.uiRtStat.0 := p_tyMcParamCurr.bAIVSizeDisabled;
	tyP0205OpsAIV.tyIOMonitor.tyBitmapMagSLarge3.uiRtStat.0 := p_tyMcParamCurr.bAIVSizeDisabled;
	tyP0205OpsAIV.tyIOMonitor.tyBitmapMagSLarge4.uiRtStat.0 := p_tyMcParamCurr.bAIVSizeDisabled;

	CASE p_tyMcParamCurr.eAGVComProtocol OF
		McSetAGVCommOPCUA:
			tyP0205OpsAIV.tyIOMonitor.tyTxtAIVCommProtocol.usiValueIdx := 0;

		McSetAGVCommHardIO:
			tyP0205OpsAIV.tyIOMonitor.tyTxtAIVCommProtocol.usiValueIdx := 1;

		McSetAGVCommDisabled:
			tyP0205OpsAIV.tyIOMonitor.tyTxtAIVCommProtocol.usiValueIdx := 2;
	END_CASE

	tyP0205OpsAIV.tyIOMonitor.tyBtnMESActive.uiRtStat.0 := p_tyMcParamCurr.eAGVComProtocol <> 0;
END_ACTION
```

#### Act_OptP0205IOMonitor.st
```iecst
ACTION Act_OptP0205IOMonitor:

	//Digital Input
	//AIV Err
	IF p_tyDI.bSOT1AIVError THEN
		tyP0205OpsAIV.tyIOMonitor.tyBitmapAIVErr1.usiValueIdx		:= 2;
	ELSE
		tyP0205OpsAIV.tyIOMonitor.tyBitmapAIVErr1.usiValueIdx		:= 0;
	END_IF

	IF p_tyDI.bSOT2AIVError THEN
		tyP0205OpsAIV.tyIOMonitor.tyBitmapAIVErr2.usiValueIdx		:= 2;
	ELSE
		tyP0205OpsAIV.tyIOMonitor.tyBitmapAIVErr2.usiValueIdx		:= 0;
	END_IF

	IF p_tyDI.bSOT3AIVError THEN
		tyP0205OpsAIV.tyIOMonitor.tyBitmapAIVErr3.usiValueIdx		:= 2;
	ELSE
		tyP0205OpsAIV.tyIOMonitor.tyBitmapAIVErr3.usiValueIdx		:= 0;
	END_IF

	IF p_tyDI.bSOT4AIVError THEN
		tyP0205OpsAIV.tyIOMonitor.tyBitmapAIVErr4.usiValueIdx		:= 2;
	ELSE
		tyP0205OpsAIV.tyIOMonitor.tyBitmapAIVErr4.usiValueIdx		:= 0;
	END_IF

	//AIV Ready
	IF p_tyDI.bSOT1AIVReady THEN
		tyP0205OpsAIV.tyIOMonitor.tyBitmapAIVRdy1.usiValueIdx		:= 1;
	ELSE
		tyP0205OpsAIV.tyIOMonitor.tyBitmapAIVRdy1.usiValueIdx		:= 0;
	END_IF

	IF p_tyDI.bSOT2AIVReady THEN
		tyP0205OpsAIV.tyIOMonitor.tyBitmapAIVRdy2.usiValueIdx		:= 1;
	ELSE
		tyP0205OpsAIV.tyIOMonitor.tyBitmapAIVRdy2.usiValueIdx		:= 0;
	END_IF

	IF p_tyDI.bSOT3AIVReady THEN
		tyP0205OpsAIV.tyIOMonitor.tyBitmapAIVRdy3.usiValueIdx		:= 1;
	ELSE
		tyP0205OpsAIV.tyIOMonitor.tyBitmapAIVRdy3.usiValueIdx		:= 0;
	END_IF

	IF p_tyDI.bSOT4AIVReady THEN
		tyP0205OpsAIV.tyIOMonitor.tyBitmapAIVRdy4.usiValueIdx		:= 1;
	ELSE
		tyP0205OpsAIV.tyIOMonitor.tyBitmapAIVRdy4.usiValueIdx		:= 0;
	END_IF

	//AIV Available
	IF p_tyDI.bSOT1AIVAvailable THEN
		tyP0205OpsAIV.tyIOMonitor.tyBitmapAIVAvail1.usiValueIdx		:= 1;
	ELSE
		tyP0205OpsAIV.tyIOMonitor.tyBitmapAIVAvail1.usiValueIdx		:= 0;
	END_IF

	IF p_tyDI.bSOT2AIVAvailable THEN
		tyP0205OpsAIV.tyIOMonitor.tyBitmapAIVAvail2.usiValueIdx		:= 1;
	ELSE
		tyP0205OpsAIV.tyIOMonitor.tyBitmapAIVAvail2.usiValueIdx		:= 0;
	END_IF

	IF p_tyDI.bSOT3AIVAvailable THEN
		tyP0205OpsAIV.tyIOMonitor.tyBitmapAIVAvail3.usiValueIdx		:= 1;
	ELSE
		tyP0205OpsAIV.tyIOMonitor.tyBitmapAIVAvail3.usiValueIdx		:= 0;
	END_IF

	IF p_tyDI.bSOT4AIVAvailable THEN
		tyP0205OpsAIV.tyIOMonitor.tyBitmapAIVAvail4.usiValueIdx		:= 1;
	ELSE
		tyP0205OpsAIV.tyIOMonitor.tyBitmapAIVAvail4.usiValueIdx		:= 0;
	END_IF

	//AIV Size
	IF p_tyDI.bSOT1AIVSizeLarge THEN
		tyP0205OpsAIV.tyIOMonitor.tyBitmapAIVSLarge1.usiValueIdx		:= 1;
	ELSE
		tyP0205OpsAIV.tyIOMonitor.tyBitmapAIVSLarge1.usiValueIdx		:= 0;
	END_IF

	IF p_tyDI.bSOT2AIVSizeLarge THEN
		tyP0205OpsAIV.tyIOMonitor.tyBitmapAIVSLarge2.usiValueIdx		:= 1;
	ELSE
		tyP0205OpsAIV.tyIOMonitor.tyBitmapAIVSLarge2.usiValueIdx		:= 0;
	END_IF

	IF p_tyDI.bSOT3AIVSizeLarge THEN
		tyP0205OpsAIV.tyIOMonitor.tyBitmapAIVSLarge3.usiValueIdx		:= 1;
	ELSE
		tyP0205OpsAIV.tyIOMonitor.tyBitmapAIVSLarge3.usiValueIdx		:= 0;
	END_IF

	IF p_tyDI.bSOT4AIVSizeLarge THEN
		tyP0205OpsAIV.tyIOMonitor.tyBitmapAIVSLarge4.usiValueIdx		:= 1;
	ELSE
		tyP0205OpsAIV.tyIOMonitor.tyBitmapAIVSLarge4.usiValueIdx		:= 0;
	END_IF

	tyP0205OpsAIV.tyIOMonitor.tyBtnAIVSotRCVOk1.bValue			:= p_tyDI.bSOT1Receive;
	tyP0205OpsAIV.tyIOMonitor.tyBtnAIVSotRCVOk2.bValue			:= p_tyDI.bSOT2Receive;
	tyP0205OpsAIV.tyIOMonitor.tyBtnAIVSotRCVOk3.bValue			:= p_tyDI.bSOT3Receive;
	tyP0205OpsAIV.tyIOMonitor.tyBtnAIVSotRCVOk4.bValue			:= p_tyDI.bSOT4Receive;

	//Digital Output
	//Mag Error
	IF p_tyDO.bSOT1MagError THEN
		tyP0205OpsAIV.tyIOMonitor.tyBitmapMagErr1.usiValueIdx		:= 2;
	ELSE
		tyP0205OpsAIV.tyIOMonitor.tyBitmapMagErr1.usiValueIdx		:= 0;
	END_IF

	IF p_tyDO.bSOT2MagError THEN
		tyP0205OpsAIV.tyIOMonitor.tyBitmapMagErr2.usiValueIdx		:= 2;
	ELSE
		tyP0205OpsAIV.tyIOMonitor.tyBitmapMagErr2.usiValueIdx		:= 0;
	END_IF

	IF p_tyDO.bSOT3MagError THEN
		tyP0205OpsAIV.tyIOMonitor.tyBitmapMagErr3.usiValueIdx		:= 2;
	ELSE
		tyP0205OpsAIV.tyIOMonitor.tyBitmapMagErr3.usiValueIdx		:= 0;
	END_IF

	IF p_tyDO.bSOT4MagError THEN
		tyP0205OpsAIV.tyIOMonitor.tyBitmapMagErr4.usiValueIdx		:= 2;
	ELSE
		tyP0205OpsAIV.tyIOMonitor.tyBitmapMagErr4.usiValueIdx		:= 0;
	END_IF

	//Mag Ready
	IF p_tyDO.bSOT1MagReady THEN
		tyP0205OpsAIV.tyIOMonitor.tyBitmapMagRdy1.usiValueIdx		:= 1;
	ELSE
		tyP0205OpsAIV.tyIOMonitor.tyBitmapMagRdy1.usiValueIdx		:= 0;
	END_IF

	IF p_tyDO.bSOT2MagReady THEN
		tyP0205OpsAIV.tyIOMonitor.tyBitmapMagRdy2.usiValueIdx		:= 1;
	ELSE
		tyP0205OpsAIV.tyIOMonitor.tyBitmapMagRdy2.usiValueIdx		:= 0;
	END_IF

	IF p_tyDO.bSOT3MagReady THEN
		tyP0205OpsAIV.tyIOMonitor.tyBitmapMagRdy3.usiValueIdx		:= 1;
	ELSE
		tyP0205OpsAIV.tyIOMonitor.tyBitmapMagRdy3.usiValueIdx		:= 0;
	END_IF

	IF p_tyDO.bSOT4MagReady THEN
		tyP0205OpsAIV.tyIOMonitor.tyBitmapMagRdy4.usiValueIdx		:= 1;
	ELSE
		tyP0205OpsAIV.tyIOMonitor.tyBitmapMagRdy4.usiValueIdx		:= 0;
	END_IF

	//Mag Available
	IF p_tyDO.bSOT1MagAvailable THEN
		tyP0205OpsAIV.tyIOMonitor.tyBitmapMagAvail1.usiValueIdx		:= 1;
	ELSE
		tyP0205OpsAIV.tyIOMonitor.tyBitmapMagAvail1.usiValueIdx		:= 0;
	END_IF

	IF p_tyDO.bSOT2MagAvailable THEN
		tyP0205OpsAIV.tyIOMonitor.tyBitmapMagAvail2.usiValueIdx		:= 1;
	ELSE
		tyP0205OpsAIV.tyIOMonitor.tyBitmapMagAvail2.usiValueIdx		:= 0;
	END_IF

	IF p_tyDO.bSOT3MagAvailable THEN
		tyP0205OpsAIV.tyIOMonitor.tyBitmapMagAvail3.usiValueIdx		:= 1;
	ELSE
		tyP0205OpsAIV.tyIOMonitor.tyBitmapMagAvail3.usiValueIdx		:= 0;
	END_IF

	IF p_tyDO.bSOT4MagAvailable THEN
		tyP0205OpsAIV.tyIOMonitor.tyBitmapMagAvail4.usiValueIdx		:= 1;
	ELSE
		tyP0205OpsAIV.tyIOMonitor.tyBitmapMagAvail4.usiValueIdx		:= 0;
	END_IF

	//Mag Size
	IF p_tyDO.bSOT1MagSizeLarge THEN
		tyP0205OpsAIV.tyIOMonitor.tyBitmapMagSLarge1.usiValueIdx		:= 1;
	ELSE
		tyP0205OpsAIV.tyIOMonitor.tyBitmapMagSLarge1.usiValueIdx		:= 0;
	END_IF

	IF p_tyDO.bSOT2MagSizeLarge THEN
		tyP0205OpsAIV.tyIOMonitor.tyBitmapMagSLarge2.usiValueIdx		:= 1;
	ELSE
		tyP0205OpsAIV.tyIOMonitor.tyBitmapMagSLarge2.usiValueIdx		:= 0;
	END_IF

	IF p_tyDO.bSOT3MagSizeLarge THEN
		tyP0205OpsAIV.tyIOMonitor.tyBitmapMagSLarge3.usiValueIdx		:= 1;
	ELSE
		tyP0205OpsAIV.tyIOMonitor.tyBitmapMagSLarge3.usiValueIdx		:= 0;
	END_IF

	IF p_tyDO.bSOT4MagSizeLarge THEN
		tyP0205OpsAIV.tyIOMonitor.tyBitmapMagSLarge4.usiValueIdx		:= 1;
	ELSE
		tyP0205OpsAIV.tyIOMonitor.tyBitmapMagSLarge4.usiValueIdx		:= 0;
	END_IF

	//MES Name
	tyP0205OpsAIV.tyIOMonitor.tyStringMesName.sValue			:= p_tyTagFromMes.sMESName;
	CASE p_tyMcParamCurr.eAGVComProtocol OF
		McSetAGVCommOPCUA:
			//Req To Bring
			tyP0205OpsAIV.tyIOMonitor.tyBtnReqAIVToBring1.bValue		:= p_tyTagToMes.tyTagStatOfPlatforms[1].bReqAIVToBring;
			tyP0205OpsAIV.tyIOMonitor.tyBtnReqAIVToBring2.bValue		:= p_tyTagToMes.tyTagStatOfPlatforms[2].bReqAIVToBring;
			tyP0205OpsAIV.tyIOMonitor.tyBtnReqAIVToBring3.bValue		:= p_tyTagToMes.tyTagStatOfPlatforms[3].bReqAIVToBring;
			tyP0205OpsAIV.tyIOMonitor.tyBtnReqAIVToBring4.bValue		:= p_tyTagToMes.tyTagStatOfPlatforms[4].bReqAIVToBring;
			//Req To Get
			tyP0205OpsAIV.tyIOMonitor.tyBtnReqAIVToGet1.bValue		:= p_tyTagToMes.tyTagStatOfPlatforms[1].bReqAIVToGet;
			tyP0205OpsAIV.tyIOMonitor.tyBtnReqAIVToGet2.bValue		:= p_tyTagToMes.tyTagStatOfPlatforms[2].bReqAIVToGet;
			tyP0205OpsAIV.tyIOMonitor.tyBtnReqAIVToGet3.bValue		:= p_tyTagToMes.tyTagStatOfPlatforms[3].bReqAIVToGet;
			tyP0205OpsAIV.tyIOMonitor.tyBtnReqAIVToGet4.bValue		:= p_tyTagToMes.tyTagStatOfPlatforms[4].bReqAIVToGet;

			tyP0205OpsAIV.tyIOMonitor.tyBtnMESActive.bValue				:= p_tyTagFromMes.bActive;
		McSetAGVCommHardIO:
			//Req To Bring
			tyP0205OpsAIV.tyIOMonitor.tyBtnReqAIVToBring1.bValue		:= p_tyDO.bMag1ReqToBring;
			tyP0205OpsAIV.tyIOMonitor.tyBtnReqAIVToBring2.bValue		:= p_tyDO.bMag2ReqToBring;
			tyP0205OpsAIV.tyIOMonitor.tyBtnReqAIVToBring3.bValue		:= p_tyDO.bMag3ReqToBring;
			tyP0205OpsAIV.tyIOMonitor.tyBtnReqAIVToBring4.bValue		:= p_tyDO.bMag4ReqToBring;
			//Req To Get
			tyP0205OpsAIV.tyIOMonitor.tyBtnReqAIVToGet1.bValue		:= p_tyDO.bMag1ReqToGet;
			tyP0205OpsAIV.tyIOMonitor.tyBtnReqAIVToGet2.bValue		:= p_tyDO.bMag2ReqToGet;
			tyP0205OpsAIV.tyIOMonitor.tyBtnReqAIVToGet3.bValue		:= p_tyDO.bMag3ReqToGet;
			tyP0205OpsAIV.tyIOMonitor.tyBtnReqAIVToGet4.bValue		:= p_tyDO.bMag4ReqToGet;

			tyP0205OpsAIV.tyIOMonitor.tyBtnMESActive.bValue				:= p_tyDI.bFleetManagerReady;
		McSetAGVCommDisabled:
			//Req To Bring
			tyP0205OpsAIV.tyIOMonitor.tyBtnReqAIVToBring1.bValue		:= FALSE;
			tyP0205OpsAIV.tyIOMonitor.tyBtnReqAIVToBring2.bValue		:= FALSE;
			tyP0205OpsAIV.tyIOMonitor.tyBtnReqAIVToBring3.bValue		:= FALSE;
			tyP0205OpsAIV.tyIOMonitor.tyBtnReqAIVToBring4.bValue		:= FALSE;
			//Req To Get
			tyP0205OpsAIV.tyIOMonitor.tyBtnReqAIVToGet1.bValue		:= FALSE;
			tyP0205OpsAIV.tyIOMonitor.tyBtnReqAIVToGet2.bValue		:= FALSE;
			tyP0205OpsAIV.tyIOMonitor.tyBtnReqAIVToGet3.bValue		:= FALSE;
			tyP0205OpsAIV.tyIOMonitor.tyBtnReqAIVToGet4.bValue		:= FALSE;

			tyP0205OpsAIV.tyIOMonitor.tyBtnMESActive.bValue	:= FALSE;
	END_CASE

END_ACTION
```

#### Act_EntP0206Disp.st
```iecst
ACTION Act_EntP0206Disp:

	//Access Address
	p_tyC0004Navi ACCESS ADR(tyP0206OpsMag4.tyNaviBack);

	p_tyC0005Main ACCESS ADR(tyCommon.tyMain);

	p_tyC0007Notif ACCESS ADR(tyCommon.tyNotif);

	p_tyC0008MsgBox ACCESS ADR(tyP0206OpsMag4.tyMsgBoxHide);

	p_tyC0009Info ACCESS ADR(tyCommon.tyInfo);

	p_tyC0011RcpPopUp ACCESS ADR(tyP0206OpsMag4.tyRcpPopUp);

	p_tyP0206Ops ACCESS ADR(tyP0206OpsMag4.tyOps);
	p_tyP0206IOMonitor ACCESS ADR(tyP0206OpsMag4.tyIOMonitor);
	p_tyP0206BypsInitConv ACCESS ADR(tyP0206OpsMag4.tyBypsInitConv);
	p_tyP0206Param ACCESS ADR(tyP0206OpsMag4.tyParam);

	//Display
	fUIInRtStatHide(ADR(tyP0206OpsMag4.tyIOMonitor.tyLyr.uiRtStat));
	fUIInRtStatHide(ADR(tyP0206OpsMag4.tyParam.tyLyr.uiRtStat));

	tyP0206OpsMag4.tyOps.tyBtnChgParam.uiRtStat.0	:= NOT(p_tyMcParamCurr.bChgParamEn);
	tyP0206OpsMag4.tyParam.tyNumMaxSlt.diValueMax	:= p_tyMagRcpCurrRcp.diTtlSlt;

	IF p_tyNtParamCurr.bMagAutoVerifyPrep = FALSE THEN
		tyP0206OpsMag4.tyIOMonitor.tyBtnMag4FixedClmpRS.usiTxtIdx	:= 6;
		tyP0206OpsMag4.tyIOMonitor.tyBtnMag4FixedUnclmpRS.usiTxtIdx:= 6;
		tyP0206OpsMag4.tyIOMonitor.tyBtnMag4RmtClmpRS.usiTxtIdx	:= 4;
		tyP0206OpsMag4.tyIOMonitor.tyBtnMag4RmtUnclmpRS.usiTxtIdx:= 4;
		tyP0206OpsMag4.tyIOMonitor.tyBtnMag4FixedClampCtrl.usiTxtIdx:= 0;
		tyP0206OpsMag4.tyIOMonitor.tyBtnMag4RemoteClampCtrl.usiTxtIdx:= 8;
	ELSE
		tyP0206OpsMag4.tyIOMonitor.tyBtnMag4FixedClmpRS.usiTxtIdx	:= 6;
		tyP0206OpsMag4.tyIOMonitor.tyBtnMag4FixedUnclmpRS.usiTxtIdx:= 6;
		tyP0206OpsMag4.tyIOMonitor.tyBtnMag4RmtClmpRS.usiTxtIdx	:= 4;
		tyP0206OpsMag4.tyIOMonitor.tyBtnMag4RmtUnclmpRS.usiTxtIdx:= 4;
		tyP0206OpsMag4.tyIOMonitor.tyBtnMag4FixedClampCtrl.usiTxtIdx:= 0;
		tyP0206OpsMag4.tyIOMonitor.tyBtnMag4RemoteClampCtrl.usiTxtIdx:= 8;

	END_IF

	fUIInRtStatHide(ADR(tyP0206OpsMag4.tyOps.tyBtnAIVWifi.uiRtStat));
	fUIInRtStatHide(ADR(tyP0206OpsMag4.tyOps.tyTxtLblAIV.uiRtStat));
END_ACTION
```

#### Act_OptP0206Navi.st
```iecst
ACTION Act_OptP0206Navi:

	IF tyP0206OpsMag4.tyNaviBack.tyBtnBack.bRtCompl = TRUE THEN
		tyP0206OpsMag4.tyNaviBack.tyBtnBack.bRtCompl	:= FALSE;
		tyP0206OpsMag4.tyNaviBack.tyBtnBack.bValue		:= FALSE;

		eChgPage	:= UIP0200OpsGen;

	END_IF

END_ACTION
```

#### Act_OptP0206ChgPage.st
```iecst
ACTION Act_OptP0206ChgPage:

	IF tyP0206OpsMag4.tyOps.tyHotspotMagInfo.bRtCompl = TRUE THEN
		tyP0206OpsMag4.tyOps.tyHotspotMagInfo.bRtCompl	:= FALSE;

		eChgPage	:= UIP0800MagInfo;
		bDisplayMag4Info := TRUE;
	END_IF

END_ACTION
```

#### Act_OptP0206UpdtDat.st
```iecst
ACTION Act_OptP0206UpdtDat:

	//Status
	fbMcStatUpdtTm(IN := TRUE);
	IF fbMcStatUpdtTm.Q = TRUE THEN
		fbMcStatUpdtTm(IN := FALSE);

		IF p_tyNtParamCurr.bProjLifterMagPlatform THEN
			tyP0206OpsMag4.tyOps.tyStringMcStat.sValue	:= p_sOpsLifMagLDStepTxt;
		ELSE
			tyP0206OpsMag4.tyOps.tyStringMcStat.sValue	:= p_sOpsMagConvLD4StepTxt;
		END_IF

	END_IF

	//Mode
	tyP0206OpsMag4.tyOps.tyTxtMod.usiValueIdx	:= p_tyProdRcpCurrRcp1.usiMcMod;

	//Width
	IF p_tyNtParamCurr.bAWPrep = TRUE AND p_tyMcParamCurr.bAWDis = FALSE THEN
		tyP0206OpsMag4.tyOps.tyNumWidth.diValue	:= p_tyMcParamCurr.diWidthAtHmPosInUM - p_diAWOpenActualPos;
		tyP0206OpsMag4.tyOps.tyNumWidth2.diValue	:= p_tyMcParamCurr.diWidthAtHmPosInUM - p_diAWOpenActualPos;
	ELSE
		tyP0206OpsMag4.tyOps.tyNumWidth.diValue	:= p_tyProdRcpCurrRcp1.diWidthInUM;
		tyP0206OpsMag4.tyOps.tyNumWidth2.diValue	:= p_tyProdRcpCurrRcp1.diWidthInUM2;
	END_IF

	//Program Info
	IF p_tyNtParamCurr.eProjMag <> LDMagQuadruple THEN
		tyP0206OpsMag4.tyOps.tyStringProdNm.sValue		:= p_tyProdRcpCurrRcp2.sRcpNm;
		tyP0206OpsMag4.tyOps.tyNumMinSltRange.diValue		:= p_tyProdRcpCurrRcp2.diMinSltValue;
		tyP0206OpsMag4.tyOps.tyNumMaxSltRange.diValue		:= p_tyProdRcpCurrRcp2.diMaxSltValue;
		tyP0206OpsMag4.tyOps.tyBtnToptoBtm.bValue			:= p_tyProdRcpCurrRcp2.bTopToBtm;
		tyP0206OpsMag4.tyOps.tyNumPitch.diValue			:= p_tyProdRcpCurrRcp2.diPitch;
		//Magazine Info
		tyP0206OpsMag4.tyOps.tyStringMagNm.sValue	:= p_tyMagRcpCurrRcp.sRcpNm;
	ELSE
		CASE p_tyProdRcpCurrRcp2.usiMcMod OF
			0:
				tyP0206OpsMag4.tyOps.tyStringProdNm.sValue		:= p_tyProdRcpCurrRcp2.sRcpNm;
				tyP0206OpsMag4.tyOps.tyNumMinSltRange.diValue		:= p_tyProdRcpCurrRcp2.diMinSltValue;
				tyP0206OpsMag4.tyOps.tyNumMaxSltRange.diValue		:= p_tyProdRcpCurrRcp2.diMaxSltValue;
				tyP0206OpsMag4.tyOps.tyBtnToptoBtm.bValue			:= p_tyProdRcpCurrRcp2.bTopToBtm;
				tyP0206OpsMag4.tyOps.tyNumPitch.diValue			:= p_tyProdRcpCurrRcp2.diPitch;
				//Magazine Info
				tyP0206OpsMag4.tyOps.tyStringMagNm.sValue	:= p_tyMagRcpCurrRcp.sRcpNm;
			1,2:

				tyP0206OpsMag4.tyOps.tyStringProdNm.sValue		:= p_tyProdRcpCurrRcp2.sRcpNm;
				tyP0206OpsMag4.tyOps.tyNumMinSltRange.diValue		:= p_tyProdRcpCurrRcp2.diMinSltValueRear;
				tyP0206OpsMag4.tyOps.tyNumMaxSltRange.diValue		:= p_tyProdRcpCurrRcp2.diMaxSltValueRear;
				tyP0206OpsMag4.tyOps.tyBtnToptoBtm.bValue			:= p_tyProdRcpCurrRcp2.bTopToBtm;
				tyP0206OpsMag4.tyOps.tyNumPitch.diValue			:= p_tyProdRcpCurrRcp2.diPitchRear;
				//Magazine Info
				tyP0206OpsMag4.tyOps.tyStringMagNm.sValue	:= p_tyMagRcpCurrRcp1.sRcpNm;
		END_CASE
	END_IF
	//Magazine Info
//	tyP0206OpsMag4.tyOps.tyStringMagNm.sValue	:= p_tyMagRcpCurrRcp.sRcpNm;

	IF p_bBuffer4MagPresent = TRUE THEN
		tyP0206OpsMag4.tyOps.tyNumMag4AvlQty.diValue	:= p_tyBuffer4BffrStat.diTtlGdBrd + p_tyBuffer4BffrStat.diTtlBadBrd;
		tyP0206OpsMag4.tyOps.tyNumMag4TtlSlt.diValue	:= p_tyBuffer4BffrStat.diTtlBrdCap;
	ELSE
		tyP0206OpsMag4.tyOps.tyNumMag4AvlQty.diValue	:= 0;
		tyP0206OpsMag4.tyOps.tyNumMag4TtlSlt.diValue	:= 0;
	END_IF

	//Magazine Present States
	IF p_bBuffer4MagPresent = TRUE THEN

		IF p_tyBuffer4BffrStat.bBffrFull = TRUE THEN
			tyP0206OpsMag4.tyOps.tyTxtMag4Stat.usiValueIdx := 2;
			tyP0206OpsMag4.tyOps.tyTxtMag4Stat.usiColor	   := 0;
		ELSIF p_tyBuffer4BffrStat.bBffrMty = TRUE THEN
			tyP0206OpsMag4.tyOps.tyTxtMag4Stat.usiValueIdx := 1;
			tyP0206OpsMag4.tyOps.tyTxtMag4Stat.usiColor	   := 1;
		ELSE
			tyP0206OpsMag4.tyOps.tyTxtMag4Stat.usiValueIdx := 3;
			tyP0206OpsMag4.tyOps.tyTxtMag4Stat.usiColor	   := 0;
		END_IF

	ELSE
		tyP0206OpsMag4.tyOps.tyTxtMag4Stat.usiValueIdx := 0;
		tyP0206OpsMag4.tyOps.tyTxtMag4Stat.usiColor	   := 1;
	END_IF

	//Product Recipe 254
	tyP0206OpsMag4.tyOps.tyHotspotShowLRcp.uiRtStat.0 := NOT(tyP0206OpsMag4.tyOps.tyStringProdNm.sValue <> '');

	IF tyP0206OpsMag4.tyOps.tyHotspotShowLRcp.bRtCompl = TRUE THEN
		tyP0206OpsMag4.tyOps.tyHotspotShowLRcp.bRtCompl := FALSE;

		fUIInRtStatOff(ADR(tyP0206OpsMag4.tyRcpPopUp.tyLyr.uiRtStat));

		tyP0206OpsMag4.tyRcpPopUp.tyStringInfo.sValue  := p_tyProdRcpCurrRcp1.sRcpNm;

	ELSIF tyP0206OpsMag4.tyRcpPopUp.tyHotspotClose.bRtCompl = TRUE THEN
		tyP0206OpsMag4.tyRcpPopUp.tyHotspotClose.bRtCompl := FALSE;

		fUIInRtStatHide(ADR(tyP0206OpsMag4.tyRcpPopUp.tyLyr.uiRtStat));

	END_IF
END_ACTION
```

#### Act_OptP0206IOMonitor.st
```iecst
ACTION Act_OptP0206IOMonitor:

	IF tyP0206OpsMag4.tyOps.tyHotspotIOMonitor.bRtCompl = TRUE THEN
		tyP0206OpsMag4.tyOps.tyHotspotIOMonitor.bRtCompl	:= FALSE;

		fUIInRtStatOff(ADR(tyP0206OpsMag4.tyIOMonitor.tyLyr.uiRtStat));

		p_tyC0004Navi ACCESS ADR(tyP0206OpsMag4.tyNaviHide);

	ELSIF tyP0206OpsMag4.tyIOMonitor.tyHotspotClose.bRtCompl = TRUE THEN
		tyP0206OpsMag4.tyIOMonitor.tyHotspotClose.bRtCompl	:= FALSE;

		fUIInRtStatHide(ADR(tyP0206OpsMag4.tyIOMonitor.tyLyr.uiRtStat));

		p_tyC0004Navi ACCESS ADR(tyP0206OpsMag4.tyNaviBack);

	END_IF

	IF tyP0206OpsMag4.tyIOMonitor.tyLyr.uiRtStat.0 = FALSE THEN

		//Digital Input
		tyP0206OpsMag4.tyIOMonitor.tyBtnSafetyRlySig.bValue				:= p_tyDI.bSafetyRlySig;
		tyP0206OpsMag4.tyIOMonitor.tyBtnEStop.bValue					:= p_tyDI.bEStopSig;
		tyP0206OpsMag4.tyIOMonitor.tyBtnCoverSWSig.bValue				:= p_tyDI.bCoverSWSig;
		tyP0206OpsMag4.tyIOMonitor.tyBtnDSBA.bValue						:= p_tyDI.bDSBA;
		tyP0206OpsMag4.tyIOMonitor.tyBtnDSBB.bValue						:= p_tyDI.bDSBB;
		tyP0206OpsMag4.tyIOMonitor.tyBtnMag4FixedClmpRS.bValue			:= p_tyDI.bMag4FixedClampRS;
		tyP0206OpsMag4.tyIOMonitor.tyBtnMag4FixedUnclmpRS.bValue		:= p_tyDI.bMag4FixedUnclampRS;
		tyP0206OpsMag4.tyIOMonitor.tyBtnMag4RmtClmpRS.bValue			:= p_tyDI.bMag4RemoteClampRS;
		tyP0206OpsMag4.tyIOMonitor.tyBtnMag4RmtUnclmpRS.bValue			:= p_tyDI.bMag4RemoteUnclampRS;
		tyP0206OpsMag4.tyIOMonitor.tyBtnMag4ConvEntrySen.bValue			:= p_tyDI.bMagConvEntSen4;
		tyP0206OpsMag4.tyIOMonitor.tyBtnMag4PresentSen.bValue			:= p_tyDI.bMagPresentSen4;
		tyP0206OpsMag4.tyIOMonitor.tyBtnMag4AIVInPosSen1.bValue			:= p_tyDI.bMag4AGVInPosSen1;
		tyP0206OpsMag4.tyIOMonitor.tyBtnMag4AIVInPosSen2.bValue			:= p_tyDI.bMag4AGVInPosSen2;
		tyP0206OpsMag4.tyIOMonitor.tyBtnMag4OrientationChkSen1.bValue	:= p_tyDI.bMag4OrientChkSen1;
		tyP0206OpsMag4.tyIOMonitor.tyBtnMag4OrientationChkSen2.bValue	:= p_tyDI.bMag4OrientChkSen2;

		tyP0206OpsMag4.tyIOMonitor.tyBtnSelUnclampRS.bValue				:= p_tyDI.bMag4SelUnClampRS;

		tyP0206OpsMag4.tyIOMonitor.tyBtnCAB717Sen.bValue				:= p_tyDI.bMagConvCAB717MagSen4;
		tyP0206OpsMag4.tyIOMonitor.tyBtnHeightSen.bValue				:= p_tyDI.bMagConvHeightSen4;
		tyP0206OpsMag4.tyIOMonitor.tyBtnMagSmallSen.bValue				:= p_tyDI.bMagConvSmallMagSen4;
		tyP0206OpsMag4.tyIOMonitor.tyBtnMagLargeSen.bValue				:= p_tyDI.bMagConvLargeMagSen4;

		//Digital Output
		tyP0206OpsMag4.tyIOMonitor.tyBtnSafetyRlyRst.bValue				:= p_tyDO.bSafetyRlyRst;
		tyP0206OpsMag4.tyIOMonitor.tyBtnTLGreen.bValue					:= p_tyDO.bTLGreen;
		tyP0206OpsMag4.tyIOMonitor.tyBtnTLAmber.bValue					:= p_tyDO.bTLAmber;
		tyP0206OpsMag4.tyIOMonitor.tyBtnTLRed.bValue					:= p_tyDO.bTLRed;
		tyP0206OpsMag4.tyIOMonitor.tyBtnBuzzer.bValue					:= p_tyDO.bBuzzer;
		tyP0206OpsMag4.tyIOMonitor.tyBtnDBAA.bValue						:= p_tyDO.bDBAA;
		tyP0206OpsMag4.tyIOMonitor.tyBtnDBAB.bValue						:= p_tyDO.bDBAB;
		tyP0206OpsMag4.tyIOMonitor.tyBtnMag4FixedClampCtrl.bValue		:= p_tyDO.bMag4FixedClampCtrl;
		tyP0206OpsMag4.tyIOMonitor.tyBtnMag4RemoteClampCtrl.bValue		:= p_tyDO.bMag4RemoteClampCtrl;
		tyP0206OpsMag4.tyIOMonitor.tyBtnMag4ConvMtrIn.bValue			:= p_tyDO.bMag4ConvMtrIn;
		tyP0206OpsMag4.tyIOMonitor.tyBtnMag4ConvMtrOut.bValue			:= p_tyDO.bMag4ConvMtrOut;
		tyP0206OpsMag4.tyIOMonitor.tyBtnMagSelClampCtrl.bValue			:= p_tyDO.bMag4SelClampCtrl;
	END_IF

END_ACTION
```

#### Act_OptP0206AIVDat.st
```iecst
ACTION Act_OptP0206AIVDat:

	//Show Change Mag Button only in Manual Exchane Mode
	tyP0206OpsMag4.tyOps.tyBtnChgMag.uiRtStat.0 := p_tyMcParamCurr.eMagExMode = McSetMagXcAutoMode AND p_tyMcParamCurr.eAGVComProtocol <> McSetAGVCommDisabled OR p_tyNtParamCurr.bProjLifterMagPlatform;;
	tyP0206OpsMag4.tyOps.tyBitmapChgMag.uiRtStat.0 := p_tyMcParamCurr.eMagExMode = McSetMagXcAutoMode AND p_tyMcParamCurr.eAGVComProtocol <> McSetAGVCommDisabled OR p_tyNtParamCurr.bProjLifterMagPlatform;;
	//LED Wifi
	tyP0206OpsMag4.tyOps.tyBtnAIVWifi.bValue	:= p_bAGVOnline;

	//Change Magazine
	IF p_tyNtParamCurr.bProjBtnInsertRmvMag = TRUE THEN

		IF EDGENEG(p_bOpsStatusRun) THEN
			bNewMag4	:= FALSE;
			tyP0206OpsMag4.tyOps.tyBtnChgMag.bRtLk	:= FALSE;
			tyP0206OpsMag4.tyOps.tyBtnChgMag.bRtCompl	:= FALSE;
			tyP0206OpsMag4.tyOps.tyBtnChgMag.bValue		:= FALSE;
		END_IF

		IF tyP0206OpsMag4.tyOps.tyBtnChgMag.bRtCompl = TRUE THEN
			tyP0206OpsMag4.tyOps.tyBtnChgMag.bRtCompl	:= FALSE;
			bNewMag4	:= p_bOpsMagConvLD4NewMagAllw;
			bRlsMag4	:= p_bOpsMagConvLD4RlsMagAllw;
		END_IF

		IF bNewMag4 = TRUE THEN
			tyP0206OpsMag4.tyOps.tyBitmapChgMag.usiValueIdx	:= 1;
			IF p_tyDI.bMag4FixedUnclampRS = FALSE  OR p_eMagConv2Clp4Status = Error
				THEN
				bNewMag4	:= FALSE;
				tyP0206OpsMag4.tyOps.tyBtnChgMag.bValue	:= FALSE;
				tyP0206OpsMag4.tyOps.tyBtnChgMag.bRtLk	:= FALSE;
				tyP0206OpsMag4.tyOps.tyBitmapChgMag.usiValueIdx	:= 0;
			END_IF

		ELSIF bRlsMag4 = TRUE THEN
			tyP0206OpsMag4.tyOps.tyBitmapChgMag.usiValueIdx	:= 1;
			IF(p_tyDI.bMag4FixedUnclampRS = TRUE AND p_tyDI.bMagPresentSen4 = FALSE)
				THEN
				bRlsMag4	:= FALSE;
				tyP0206OpsMag4.tyOps.tyBtnChgMag.bValue	:= FALSE;
				tyP0206OpsMag4.tyOps.tyBtnChgMag.bRtLk	:= FALSE;
				tyP0206OpsMag4.tyOps.tyBitmapChgMag.usiValueIdx	:= 0;
			END_IF

		END_IF

		IF p_tyDI.bMagPresentSen4 AND p_tyDI.bMagConvEntSen4 = FALSE THEN
			tyP0206OpsMag4.tyOps.tyBtnChgMag.usiTxtIdx	:= 1;
		ELSE
			tyP0206OpsMag4.tyOps.tyBtnChgMag.usiTxtIdx	:= 0;
		END_IF

		tyP0206OpsMag4.tyOps.tyBtnChgMag.uiMaskRtStat.0	:= p_bOpsMagConvLD4NewMagAllw OR p_bOpsMagConvLD4RlsMagAllw;// OR p_tyDI.bInShutterCloseRS;

	END_IF
END_ACTION
```

#### Act_OptP0206ChgParam.st
```iecst
ACTION Act_OptP0206ChgParam:

	tyP0206OpsMag4.tyParam.tyNumMinSlt.diValueMax		:= tyP0206OpsMag4.tyParam.tyNumMaxSlt.diValue;
	tyP0206OpsMag4.tyParam.tyNumMaxSlt.diValueMin		:= tyP0206OpsMag4.tyParam.tyNumMinSlt.diValue;
	tyP0206OpsMag4.tyParam.tyNumPitch.diValueMax		:= tyP0206OpsMag4.tyParam.tyNumMaxSlt.diValue - tyP0206OpsMag4.tyParam.tyNumMinSlt.diValue + 1;
	tyP0206OpsMag4.tyParam.tyNumPitch.diValueMin		:= 1;

	tyP0206OpsMag4.tyParam.tyNumMinSltRear.diValueMax		:= tyP0206OpsMag4.tyParam.tyNumMaxSltRear.diValue;
	tyP0206OpsMag4.tyParam.tyNumMaxSltRear.diValueMin		:= tyP0206OpsMag4.tyParam.tyNumMinSltRear.diValue;
	tyP0206OpsMag4.tyParam.tyNumPitchRear.diValueMax		:= tyP0206OpsMag4.tyParam.tyNumMaxSltRear.diValue - tyP0206OpsMag4.tyParam.tyNumMinSltRear.diValue + 1;
	tyP0206OpsMag4.tyParam.tyNumPitchRear.diValueMin		:= 1;
	//Control
	IF tyP0206OpsMag4.tyOps.tyBtnChgParam.bRtCompl = TRUE THEN
		tyP0206OpsMag4.tyOps.tyBtnChgParam.bRtCompl	:= FALSE;

		tyProdRcpCurrRcpWr	:= p_tyProdRcpCurrRcp0;

		tyP0206OpsMag4.tyParam.tyDrpDnMcMode.usiValueIdx	:= p_tyProdRcpCurrRcp0.usiMcMod;
		tyP0206OpsMag4.tyParam.tyNumMinSlt.diValue	:= p_tyProdRcpCurrRcp0.diMinSltValue;
		tyP0206OpsMag4.tyParam.tyNumMaxSlt.diValue	:= p_tyProdRcpCurrRcp0.diMaxSltValue;
		tyP0206OpsMag4.tyParam.tyNumPitch.diValue		:= p_tyProdRcpCurrRcp0.diPitch;

		tyP0206OpsMag4.tyParam.tyNumMinSltRear.diValue	:= p_tyProdRcpCurrRcp0.diMinSltValueRear;
		tyP0206OpsMag4.tyParam.tyNumMaxSltRear.diValue	:= p_tyProdRcpCurrRcp0.diMaxSltValueRear;
		tyP0206OpsMag4.tyParam.tyNumPitchRear.diValue		:= p_tyProdRcpCurrRcp0.diPitchRear;

		fUIInRtStatOff(ADR(tyP0206OpsMag4.tyParam.tyLyr.uiRtStat));

	END_IF

	tyP0206OpsMag4.tyOps.tyBtnChgParam.bValue	:= tyP0206OpsMag4.tyParam.tyLyr.uiRtStat.0 = FALSE;

	IF tyP0206OpsMag4.tyParam.tyLyr.uiRtStat.0 = FALSE THEN

		IF tyP0206OpsMag4.tyParam.tyBtnSave.bRtCompl = TRUE THEN

			tyProdRcpCurrRcpWr.usiMcMod	:= tyP0206OpsMag4.tyParam.tyDrpDnMcMode.usiValueIdx;
			tyProdRcpCurrRcpWr.diMinSltValue := tyP0206OpsMag4.tyParam.tyNumMinSlt.diValue;
			tyProdRcpCurrRcpWr.diMaxSltValue := tyP0206OpsMag4.tyParam.tyNumMaxSlt.diValue;
			tyProdRcpCurrRcpWr.diPitch := tyP0206OpsMag4.tyParam.tyNumPitch.diValue;

			tyProdRcpCurrRcpWr.diMinSltValueRear := tyP0206OpsMag4.tyParam.tyNumMinSltRear.diValue;
			tyProdRcpCurrRcpWr.diMaxSltValueRear := tyP0206OpsMag4.tyParam.tyNumMaxSltRear.diValue;
			tyProdRcpCurrRcpWr.diPitchRear := tyP0206OpsMag4.tyParam.tyNumPitchRear.diValue;

			eProdRcpAct	:= ProdRcpActWriteCurrRcpParam;

			IF p_eProdRcpStatus = Done AND p_eProdRcpStat = ProdRcpActWriteCurrRcpParam THEN
				eProdRcpAct	:= ProdRcpActIdle;

				//UIP0400
				tyP0400ProdSel.tyProdSel.tyTxtMcMode.usiValueIdx	:= p_tyProdRcpCurrRcp0.usiMcMod;

				tyP0400ProdSel.tyProdSel.tyNumMinSlt.diValue	:= p_tyProdRcpCurrRcp0.diMinSltValue;
				tyP0400ProdSel.tyProdSel.tyNumMaxSlt.diValue	:= p_tyProdRcpCurrRcp0.diMaxSltValue;
				tyP0400ProdSel.tyProdSel.tyNumPitch.diValue		:= p_tyProdRcpCurrRcp0.diPitch;

				tyP0400ProdSel.tyProdSel.tyNumMinSltRear.diValue	:= p_tyProdRcpCurrRcp0.diMinSltValueRear;
				tyP0400ProdSel.tyProdSel.tyNumMaxSltRear.diValue	:= p_tyProdRcpCurrRcp0.diMaxSltValueRear;
				tyP0400ProdSel.tyProdSel.tyNumPitchRear.diValue		:= p_tyProdRcpCurrRcp0.diPitchRear;

				tyP0206OpsMag4.tyParam.tyBtnSave.bRtCompl	:= FALSE;
				tyP0206OpsMag4.tyParam.tyBtnSave.bValue		:= FALSE;

				fUIInRtStatHide(ADR(tyP0206OpsMag4.tyParam.tyLyr.uiRtStat));

			ELSIF p_eProdRcpStatus = Error THEN
				p_tyC0008MsgBox ACCESS ADR(tyP0206OpsMag4.tyMsgBoxSaveErr);

				IF tyP0206OpsMag4.tyMsgBoxSaveErr.tyBtnNo.bRtCompl = TRUE THEN
					tyP0206OpsMag4.tyMsgBoxSaveErr.tyBtnNo.bRtCompl	:= FALSE;
					tyP0206OpsMag4.tyMsgBoxSaveErr.tyBtnNo.bValue	:= FALSE;

					p_tyC0008MsgBox ACCESS ADR(tyP0206OpsMag4.tyMsgBoxHide);

					//Restore Param
					tyProdRcpCurrRcpWr	:= p_tyProdRcpCurrRcp2;

					tyP0206OpsMag4.tyParam.tyBtnSave.bRtCompl		:= FALSE;
					tyP0206OpsMag4.tyParam.tyBtnSave.bValue			:= FALSE;

					fUIInRtStatHide(ADR(tyP0206OpsMag4.tyParam.tyLyr.uiRtStat));

				END_IF

			END_IF

		ELSIF tyP0206OpsMag4.tyParam.tyBtnCancel.bRtCompl = TRUE THEN
			tyP0206OpsMag4.tyParam.tyBtnCancel.bRtCompl				:= FALSE;
			tyP0206OpsMag4.tyParam.tyBtnCancel.bValue				:= FALSE;

			fUIInRtStatHide(ADR(tyP0206OpsMag4.tyParam.tyLyr.uiRtStat));

		END_IF

	END_IF

	//Mask
	tyP0206OpsMag4.tyOps.tyBtnChgParam.uiMaskRtStat.0	:= p_tyUsrMgmtCurrAccessRgt.bChgParam AND p_bOpsStatusStop;

END_ACTION
```

#### Act_OptP0206InsertRmvMag.st
```iecst
ACTION Act_OptP0206InsertRmvMag:

	//Insert & Removed Magazine Manually Without Button Control
//	IF p_tyNtParamCurr.bProjBtnInsertRmvMag = FALSE THEN
//
//		IF p_bOpsStatusRun AND p_bOpsMagConvLD3InitDone THEN
//
//			fbMag3EntrySenOnTm(IN := p_tyDI.bMagPresentSen3 OR p_tyDI.bMagConvEntSen3);
//
//			IF bNewMag3 = FALSE AND bRlsMag3 = FALSE THEN
//				IF p_bOpsMagConvLD3NewMagAllw AND fbMag3EntrySenOnTm.Q AND NOT p_bOpsMagConvLD3MagExitedWait THEN
//					bNewMag3	:= TRUE;
//				END_IF
//
//				IF p_bOpsMagConvLD3RlsMagAllw AND p_tyDI.bMagPresentSen3 AND p_tyDI.bInShutterCloseRS AND p_tyBuffer3BffrStat.bBffrMty THEN
//					bRlsMag3	:= TRUE;
//				END_IF
//			END_IF
//
//			IF bNewMag3 = TRUE THEN
//
//				IF p_tyDI.bMag3FixedClampRS = TRUE AND p_tyDI.bMag3RemoteClampRS = TRUE THEN
//					bNewMag3	:= FALSE;
//				END_IF
//
//			ELSIF bRlsMag3 = TRUE THEN
//
//				IF p_tyDI.bMag3FixedUnclampRS = TRUE AND p_tyDI.bMag3RemoteUnclampRS = TRUE AND p_tyDI.bMagConvEntSen3 = TRUE THEN
//					bRlsMag3	:= FALSE;
//				END_IF
//
//			END_IF
//
//		ELSE
//
//			bNewMag3	:= FALSE;
//			bRlsMag3	:= FALSE;
//
//			fbMag3EntrySenOnTm(IN := FALSE);
//
//		END_IF
//
//	END_IF

END_ACTION
```

#### Act_OptP0206RstMnl.st
```iecst
ACTION Act_OptP0206RstMnl:

	IF eCurrPage <> UIP0206OpsMag4 THEN
		bNewMag4	:= FALSE;
		bRlsMag4	:= FALSE;
		tyP0206OpsMag4.tyOps.tyBtnChgMag.bValue	:= FALSE;
		tyP0206OpsMag4.tyOps.tyBtnChgMag.bRtLk	:= FALSE;
		tyP0206OpsMag4.tyOps.tyBitmapChgMag.usiValueIdx	:= 0;
	END_IF

END_ACTION
```

#### Act_OptP0206_P0003AIVDat.st - not listed in the package file held
```iecst
ACTION Act_OptP0206_P0003AIVDat:

	//Show Change Mag Button only in Manual Exchane Mode
	tyP0206OpsMag4.tyOps.tyBtnChgMag.uiRtStat.0 := p_tyMcParamCurr.eMagExMode = McSetMagXcAutoMode AND p_tyMcParamCurr.eAGVComProtocol <> McSetAGVCommDisabled OR p_tyNtParamCurr.bProjLifterMagPlatform;;
	tyP0206OpsMag4.tyOps.tyBitmapChgMag.uiRtStat.0 := p_tyMcParamCurr.eMagExMode = McSetMagXcAutoMode AND p_tyMcParamCurr.eAGVComProtocol <> McSetAGVCommDisabled OR p_tyNtParamCurr.bProjLifterMagPlatform;;
	//LED Wifi
	tyP0206OpsMag4.tyOps.tyBtnAIVWifi.bValue	:= p_bAGVOnline;

	//Change Magazine
	IF p_tyNtParamCurr.bProjBtnInsertRmvMag = TRUE THEN

		IF EDGENEG(p_bOpsStatusRun) THEN
			bNewMag4	:= FALSE;
			tyP0206OpsMag4.tyOps.tyBtnChgMag.bRtLk	:= FALSE;
			tyP0206OpsMag4.tyOps.tyBtnChgMag.bRtCompl	:= FALSE;
			tyP0206OpsMag4.tyOps.tyBtnChgMag.bValue		:= FALSE;
		END_IF

		IF tyP0206OpsMag4.tyOps.tyBtnChgMag.bRtCompl = TRUE THEN
			tyP0206OpsMag4.tyOps.tyBtnChgMag.bRtCompl	:= FALSE;
			bNewMag4	:= p_bOpsMagConvLD4NewMagAllw;
			bRlsMag4	:= p_bOpsMagConvLD4RlsMagAllw;
		END_IF

		IF bNewMag4 = TRUE THEN
			tyP0206OpsMag4.tyOps.tyBitmapChgMag.usiValueIdx	:= 1;
			IF p_tyDI.bMag4FixedUnclampRS = FALSE  OR p_eMagConv2Clp4Status = Error
				THEN
				bNewMag4	:= FALSE;
				tyP0206OpsMag4.tyOps.tyBtnChgMag.bValue	:= FALSE;
				tyP0206OpsMag4.tyOps.tyBtnChgMag.bRtLk	:= FALSE;
				tyP0206OpsMag4.tyOps.tyBitmapChgMag.usiValueIdx	:= 0;
			END_IF

		ELSIF bRlsMag4 = TRUE THEN
			tyP0206OpsMag4.tyOps.tyBitmapChgMag.usiValueIdx	:= 1;
			IF(p_tyDI.bMag4FixedUnclampRS = TRUE AND p_tyDI.bMagPresentSen4 = FALSE)
				THEN
				bRlsMag4	:= FALSE;
				tyP0206OpsMag4.tyOps.tyBtnChgMag.bValue	:= FALSE;
				tyP0206OpsMag4.tyOps.tyBtnChgMag.bRtLk	:= FALSE;
				tyP0206OpsMag4.tyOps.tyBitmapChgMag.usiValueIdx	:= 0;
			END_IF

		END_IF

		IF p_tyDI.bMagPresentSen4 AND p_tyDI.bMagConvEntSen4 = FALSE THEN
			tyP0206OpsMag4.tyOps.tyBtnChgMag.usiTxtIdx	:= 1;
		ELSE
			tyP0206OpsMag4.tyOps.tyBtnChgMag.usiTxtIdx	:= 0;
		END_IF

		tyP0206OpsMag4.tyOps.tyBtnChgMag.uiMaskRtStat.0	:= p_bOpsMagConvLD4NewMagAllw OR p_bOpsMagConvLD4RlsMagAllw;// OR p_tyDI.bInShutterCloseRS;

	END_IF
END_ACTION
```

#### Act_EntP0300Disp.st
```iecst
ACTION Act_EntP0300Disp:

	//Access Addres
	p_tyC0005Main ACCESS ADR(tyCommon.tyMain);

	p_tyC0007Notif ACCESS ADR(tyCommon.tyNotif);

	p_tyC0008MsgBox ACCESS ADR(tyP0300McInfo.tyMsgBoxHide);

	p_tyC0009Info ACCESS ADR(tyCommon.tyInfo);

	p_tyP0300McInfo ACCESS ADR(tyP0300McInfo.tyMcInfo);

	//Display
	//Machine Name
	tyP0300McInfo.tyMcInfo.tyStringMcNm.sValue	:= p_tyMcParamCurr.sMcNm;

END_ACTION
```

#### Act_EntP0400Disp.st
```iecst
ACTION Act_EntP0400Disp:

	//Access Addres
	p_tyC0005Main ACCESS ADR(tyCommon.tyMain);

	p_tyC0007Notif ACCESS ADR(tyCommon.tyNotif);

	p_tyC0008MsgBox ACCESS ADR(tyP0400ProdSel.tyMsgBoxHide);

	p_tyC0009Info ACCESS ADR(tyCommon.tyInfo);

	p_tyC0011RcpPopUp ACCESS ADR(tyP0400ProdSel.tyRcpPopUp);

	p_tyP0400ProdSel ACCESS ADR(tyP0400ProdSel.tyProdSel);

	p_tyP0400RcpDet ACCESS ADR(tyP0400ProdSel.tyRcpDet);

	//Display
	tyP0400ProdSel.tyProdSel.tyStringSearch.bRtCompl	:= TRUE;
	tyP0400ProdSel.tyProdSel.tyStringSearch.sValue		:= '';

	fUIInRtStatHide(ADR(tyP0400ProdSel.tyRcpDet.tyLyr.uiRtStat));
	fUIInRtStatHide(ADR(tyP0400ProdSel.tyRcpDet.tyLyr1.uiRtStat));

	fUIInRtStatHide(ADR(tyP0400ProdSel.tyRcpPopUp.tyLyr.uiRtStat)); // Hide Pop Up Layer

	//Long Board
	tyP0400ProdSel.tyProdSel.tyBtnLongBrd.uiRtStat.0			:= NOT(p_tyNtParamCurr.bProjLongBrdPrep AND p_tyMcParamCurr.bLongBrdEn);
	tyP0400ProdSel.tyRcpDet.tyBtnLongBrd.uiRtStat.0				:= NOT(p_tyNtParamCurr.bProjLongBrdPrep AND p_tyMcParamCurr.bLongBrdEn);

	//Product Selection
	tyP0400ProdSel.tyProdSel.tyStringRecipeNm.sValue		:= p_tyProdRcpCurrRcp0.sRcpNm;
	tyP0400ProdSel.tyProdSel.tyNumProdWidth.diValue			:= p_tyProdRcpCurrRcp0.diWidthInUM;
	tyP0400ProdSel.tyProdSel.tyNumProdWidth2.diValue		:= p_tyProdRcpCurrRcp0.diWidthInUM2;
	tyP0400ProdSel.tyProdSel.tyNumProdWidthRear.diValue		:= p_tyProdRcpCurrRcp0.diWidthInUMRear;
	tyP0400ProdSel.tyProdSel.tyNumMaxSlt.diValue			:= p_tyProdRcpCurrRcp0.diMaxSltValue;
	tyP0400ProdSel.tyProdSel.tyNumMinSlt.diValue			:= p_tyProdRcpCurrRcp0.diMinSltValue;
	tyP0400ProdSel.tyProdSel.tyNumPitch.diValue				:= p_tyProdRcpCurrRcp0.diPitch;
	tyP0400ProdSel.tyProdSel.tyBtnToptoBtm.bValue			:= p_tyProdRcpCurrRcp0.bTopToBtm;
	tyP0400ProdSel.tyProdSel.tyBtnLongBrd.bValue			:= p_tyProdRcpCurrRcp0.bLongBrd;
	tyP0400ProdSel.tyProdSel.tyTxtMcMode.usiValueIdx		:= p_tyProdRcpCurrRcp0.usiMcMod;
	tyP0400ProdSel.tyProdSel.tyTxtFlippedBrd.usiValueIdx	:= p_tyProdRcpCurrRcp0.usiFlippedBrd;
	tyP0400ProdSel.tyProdSel.tyNumMtrPshrExtSpd.diValue		:= p_tyProdRcpCurrRcp0.diMtrPshrExtSpd;
	tyP0400ProdSel.tyProdSel.tyNumMtrPshrExtTorq.diValue	:= p_tyProdRcpCurrRcp0.diMtrPshrExtTorq;
	tyP0400ProdSel.tyProdSel.tyNumPshrOffset.diValue		:= p_tyProdRcpCurrRcp0.diPshrOffset;

END_ACTION
```

#### Act_OptP0400Load.st
```iecst
ACTION Act_OptP0400Load:

	IF tyP0400ProdSel.tyProdSel.tyBtnLoad.bRtCompl = TRUE THEN

		IF usiSelProdRcpStep = 0 THEN
			//Message Confirmation Ask - Load Product Recipe
			//Mask
			tyP0400ProdSel.tyProdSel.tyTableRecipe.uiMaskRtStat		:= FALSE;
			tyP0400ProdSel.tyProdSel.tyStringSearch.uiMaskRtStat	:= FALSE;

			p_tyC0008MsgBox ACCESS ADR(tyP0400ProdSel.tyMsgBoxSelRcpAsk);

			IF tyP0400ProdSel.tyMsgBoxSelRcpAsk.tyBtnYes.bRtCompl = TRUE THEN
				tyP0400ProdSel.tyMsgBoxSelRcpAsk.tyBtnYes.bRtCompl	:= FALSE;
				tyP0400ProdSel.tyMsgBoxSelRcpAsk.tyBtnYes.bValue	:= FALSE;

				p_tyC0008MsgBox ACCESS ADR(tyP0400ProdSel.tyMsgBoxHide);

				usiSelProdRcpStep	:= 1;

			ELSIF tyP0400ProdSel.tyMsgBoxSelRcpAsk.tyBtnNo.bRtCompl = TRUE THEN
				tyP0400ProdSel.tyMsgBoxSelRcpAsk.tyBtnNo.bRtCompl	:= FALSE;
				tyP0400ProdSel.tyMsgBoxSelRcpAsk.tyBtnNo.bValue		:= FALSE;

				p_tyC0008MsgBox ACCESS ADR(tyP0400ProdSel.tyMsgBoxHide);

				usiSelProdRcpStep	:= 99;

			END_IF

		ELSIF usiSelProdRcpStep = 1 THEN
			//Load Product Recipe
			tyProdRcpInfoIn.sRcpNm		:= tyP0400ProdSel.tyProdSel.tyTableRecipe.a_tyStringDataCol1[tyP0400Table.uiSelectedRow].sValue;

			eProdRcpAct					:= ProdRcpActLoadRcp;

			IF p_eProdRcpStat = ProdRcpActLoadRcp AND p_eProdRcpStatus = Done THEN
				eProdRcpAct				:= ProdRcpActIdle;

				IF p_bProdRcpNmEmpty = TRUE AND p_bProdRcpNmNotExist = TRUE THEN
					usiSelProdRcpStep	:= 2;
				ELSE
					//Update UI Current Recipe
					tyP0400ProdSel.tyProdSel.tyStringRecipeNm.sValue		:= p_tyProdRcpCurrRcp0.sRcpNm;
					tyP0400ProdSel.tyProdSel.tyNumProdWidth.diValue			:= p_tyProdRcpCurrRcp0.diWidthInUM;
					tyP0400ProdSel.tyProdSel.tyNumProdWidth2.diValue		:= p_tyProdRcpCurrRcp0.diWidthInUM2;
					tyP0400ProdSel.tyProdSel.tyNumMinSlt.diValue			:= p_tyProdRcpCurrRcp0.diMinSltValue;
					tyP0400ProdSel.tyProdSel.tyNumMaxSlt.diValue			:= p_tyProdRcpCurrRcp0.diMaxSltValue;
					tyP0400ProdSel.tyProdSel.tyNumPitch.diValue				:= p_tyProdRcpCurrRcp0.diPitch;
					tyP0400ProdSel.tyProdSel.tyBtnToptoBtm.bValue			:= p_tyProdRcpCurrRcp0.bTopToBtm;
					tyP0400ProdSel.tyProdSel.tyBtnLongBrd.bValue			:= p_tyProdRcpCurrRcp0.bLongBrd;
					tyP0400ProdSel.tyProdSel.tyTxtMcMode.usiValueIdx		:= p_tyProdRcpCurrRcp0.usiMcMod;
					tyP0400ProdSel.tyProdSel.tyTxtFlippedBrd.usiValueIdx	:= p_tyProdRcpCurrRcp0.usiFlippedBrd;

					tyP0400ProdSel.tyProdSel.tyNumProdWidthRear.diValue		:= p_tyProdRcpCurrRcp0.diWidthInUMRear;
					tyP0400ProdSel.tyProdSel.tyNumPitchRear.diValue			:= p_tyProdRcpCurrRcp0.diPitchRear;
					tyP0400ProdSel.tyProdSel.tyNumMinSltRear.diValue		:= p_tyProdRcpCurrRcp0.diMinSltValueRear;
					tyP0400ProdSel.tyProdSel.tyNumMaxSltRear.diValue		:= p_tyProdRcpCurrRcp0.diMaxSltValueRear;
					tyP0400ProdSel.tyProdSel.tyNumMtrPshrExtSpd.diValue		:= p_tyProdRcpCurrRcp0.diMtrPshrExtSpd;
					tyP0400ProdSel.tyProdSel.tyNumMtrPshrExtTorq.diValue	:= p_tyProdRcpCurrRcp0.diMtrPshrExtTorq;
					tyP0400ProdSel.tyProdSel.tyNumPshrOffset.diValue		:= p_tyProdRcpCurrRcp0.diPshrOffset;

					tyProdRcpCurrRcpWr	:= p_tyProdRcpCurrRcp0;

					IF ((NOT p_tyNtParamCurr.bLFUsrSetPrep AND p_tyNtParamCurr.bLeaderMc) OR (p_tyNtParamCurr.bLFUsrSetPrep AND p_tyMcParamCurr.bLFLeaderMc)) AND p_tyNtParamCurr.bLFPrep AND p_tyMcParamCurr.bLFEn AND p_tyUsrMgmtCurrAccessRgt.bLFCtrl THEN
						usiSelProdRcpStep	:= 98;
					ELSE
						usiSelProdRcpStep	:= 99;
					END_IF

				END_IF

			ELSIF p_eProdRcpStatus = Error THEN

				usiSelProdRcpStep	:= 99;

			END_IF

		ELSIF usiSelProdRcpStep = 2 THEN
			//Message Name Not Found
			p_tyC0008MsgBox ACCESS ADR(tyP0400ProdSel.tyMsgBoxSelRcpNoNm);

			IF tyP0400ProdSel.tyMsgBoxSelRcpNoNm.tyBtnNo.bRtCompl = TRUE THEN
				tyP0400ProdSel.tyMsgBoxSelRcpNoNm.tyBtnNo.bRtCompl	:= FALSE;
				tyP0400ProdSel.tyMsgBoxSelRcpNoNm.tyBtnNo.bValue	:= FALSE;

				p_tyC0008MsgBox ACCESS ADR(tyP0400ProdSel.tyMsgBoxHide);

				usiSelProdRcpStep	:= 99;

			END_IF

		ELSIF usiSelProdRcpStep = 98 THEN
			IF p_bAlarmErr AND p_tyMcAlmData.udiCode = 10000 THEN
				usiSelProdRcpStep	:= 99;
			ELSE
				//Message Confirmation Ask - Go To Leader Follower Control Page
				p_tyC0008MsgBox ACCESS ADR(tyP0400ProdSel.tyMsgBoxGoToLFCtrlAsk);
			END_IF

			IF tyP0400ProdSel.tyMsgBoxGoToLFCtrlAsk.tyBtnYes.bRtCompl = TRUE THEN
				tyP0400ProdSel.tyMsgBoxGoToLFCtrlAsk.tyBtnYes.bRtCompl	:= FALSE;
				tyP0400ProdSel.tyMsgBoxGoToLFCtrlAsk.tyBtnYes.bValue	:= FALSE;

				p_tyC0008MsgBox ACCESS ADR(tyP0400ProdSel.tyMsgBoxHide);

				eChgPage	:= UIP0700LFCtrl;

				tyCommon.tyMain.tyBtnStart.bRtCompl	:= TRUE;

				//Complete
				//Unmask
				tyP0400ProdSel.tyProdSel.tyTableRecipe.uiMaskRtStat		:= TRUE;
				tyP0400ProdSel.tyProdSel.tyStringSearch.uiMaskRtStat	:= TRUE;

				//Reset
				tyP0400ProdSel.tyProdSel.tyBtnLoad.bRtCompl	:= FALSE;
				tyP0400ProdSel.tyProdSel.tyBtnLoad.bValue	:= FALSE;

				usiSelProdRcpStep	:= 0;

			ELSIF tyP0400ProdSel.tyMsgBoxGoToLFCtrlAsk.tyBtnNo.bRtCompl = TRUE THEN
				tyP0400ProdSel.tyMsgBoxGoToLFCtrlAsk.tyBtnNo.bRtCompl	:= FALSE;
				tyP0400ProdSel.tyMsgBoxGoToLFCtrlAsk.tyBtnNo.bValue		:= FALSE;

				p_tyC0008MsgBox ACCESS ADR(tyP0400ProdSel.tyMsgBoxHide);

				usiSelProdRcpStep	:= 99;

			END_IF

		ELSIF usiSelProdRcpStep = 99 THEN
			//Complete
			//Unmask
			tyP0400ProdSel.tyProdSel.tyTableRecipe.uiMaskRtStat		:= TRUE;
			tyP0400ProdSel.tyProdSel.tyStringSearch.uiMaskRtStat	:= TRUE;

			//Reset
			tyP0400ProdSel.tyProdSel.tyBtnLoad.bRtCompl				:= FALSE;
			tyP0400ProdSel.tyProdSel.tyBtnLoad.bValue				:= FALSE;

			usiSelProdRcpStep	:= 0;

		END_IF

	END_IF

END_ACTION
```

#### Act_OptP0400Preview.st
```iecst
ACTION Act_OptP0400Preview:

	IF tyP0400ProdSel.tyProdSel.tyBtnPreview.bRtCompl = TRUE THEN

		tyProdRcpInfoIn.sRcpNm	:= tyP0400ProdSel.tyProdSel.tyTableRecipe.a_tyStringDataCol1[tyP0400Table.uiSelectedRow].sValue;

		eProdRcpAct	:= ProdRcpActGetInfo;

		IF	p_eProdRcpStat = ProdRcpActGetInfo AND p_eProdRcpStatus = Done THEN
			eProdRcpAct	:= ProdRcpActIdle;

			IF p_bProdRcpNmEmpty = TRUE AND p_bProdRcpNmNotExist = TRUE THEN
				tyP0400ProdSel.tyRcpDet.tyStringRecipeNm.sValue			:= '';
				tyP0400ProdSel.tyRcpDet.tyNumProdWidth.diValue			:= 100000;
				tyP0400ProdSel.tyRcpDet.tyNumProdWidth2.diValue			:= 100000;
				tyP0400ProdSel.tyRcpDet.tyNumProdWidthRear.diValue		:= 100000;
				tyP0400ProdSel.tyRcpDet.tyTxtMcMode.usiValueIdx			:= p_tyMcParamCurr.usiDefaultMcMod;
				tyP0400ProdSel.tyRcpDet.tyTxtFlippedBrd.usiValueIdx		:= p_tyMcParamCurr.usiDefaultFlippedBrd;
				tyP0400ProdSel.tyRcpDet.tyNumFirstSlt.diValue			:= 0;
				tyP0400ProdSel.tyRcpDet.tyNumLastSlt.diValue			:= 0;
				tyP0400ProdSel.tyRcpDet.tyNumPitch.diValue				:= 0;
				tyP0400ProdSel.tyRcpDet.tyBtnToptoBtm.bValue			:= FALSE;
				tyP0400ProdSel.tyRcpDet.tyBtnLongBrd.bValue				:= FALSE;
				tyP0400ProdSel.tyRcpDet.tyNumMtrPshrExtSpd.diValue		:= 0;
				tyP0400ProdSel.tyRcpDet.tyNumMtrPshrExtTorq.diValue		:= 0;
				tyP0400ProdSel.tyRcpDet.tyNumPshrOffset.diValue			:= p_tyProdRcpInfoOut.diPshrOffset;
			ELSE
				tyP0400ProdSel.tyRcpDet.tyStringRecipeNm.sValue			:= p_tyProdRcpInfoOut.sRcpNm;
				tyP0400ProdSel.tyRcpDet.tyNumProdWidth.diValue			:= p_tyProdRcpInfoOut.diWidthInUM;
				tyP0400ProdSel.tyRcpDet.tyNumProdWidth2.diValue			:= p_tyProdRcpInfoOut.diWidthInUM2;
				tyP0400ProdSel.tyRcpDet.tyNumProdWidthRear.diValue		:= p_tyProdRcpInfoOut.diWidthInUMRear;
				tyP0400ProdSel.tyRcpDet.tyTxtMcMode.usiValueIdx			:= p_tyProdRcpInfoOut.usiMcMod;
				tyP0400ProdSel.tyRcpDet.tyTxtFlippedBrd.usiValueIdx		:= p_tyProdRcpInfoOut.usiFlippedBrd;
				tyP0400ProdSel.tyRcpDet.tyNumFirstSlt.diValue			:= p_tyProdRcpInfoOut.diMinSltValue;
				tyP0400ProdSel.tyRcpDet.tyNumLastSlt.diValue			:= p_tyProdRcpInfoOut.diMaxSltValue;
				tyP0400ProdSel.tyRcpDet.tyNumPitch.diValue				:= p_tyProdRcpInfoOut.diPitch;
				tyP0400ProdSel.tyRcpDet.tyBtnToptoBtm.bValue			:= p_tyProdRcpInfoOut.bTopToBtm;
				tyP0400ProdSel.tyRcpDet.tyBtnLongBrd.bValue				:= p_tyProdRcpInfoOut.bLongBrd;
				tyP0400ProdSel.tyRcpDet.tyNumMtrPshrExtSpd.diValue		:= p_tyProdRcpInfoOut.diMtrPshrExtSpd;
				tyP0400ProdSel.tyRcpDet.tyNumMtrPshrExtTorq.diValue		:= p_tyProdRcpInfoOut.diMtrPshrExtTorq;
				tyP0400ProdSel.tyRcpDet.tyNumPshrOffset.diValue			:= p_tyProdRcpInfoOut.diPshrOffset;
			END_IF

			IF p_tyNtParamCurr.eProjMag = LDMagQuadruple THEN
				fUIInRtStatOff(ADR(tyP0400ProdSel.tyRcpDet.tyLyr1.uiRtStat));
			ELSE
				fUIInRtStatOff(ADR(tyP0400ProdSel.tyRcpDet.tyLyr.uiRtStat));
			END_IF
			tyP0400ProdSel.tyProdSel.tyBtnPreview.bRtCompl	:= FALSE;

		END_IF

	END_IF

	IF tyP0400ProdSel.tyRcpDet.tyHotspotClose.bRtCompl = TRUE THEN
		tyP0400ProdSel.tyRcpDet.tyHotspotClose.bRtCompl	:= FALSE;
		tyP0400ProdSel.tyProdSel.tyBtnPreview.bValue	:= FALSE;

		//Hide Recipe Details
		fUIInRtStatHide(ADR(tyP0400ProdSel.tyRcpDet.tyLyr.uiRtStat));
		fUIInRtStatHide(ADR(tyP0400ProdSel.tyRcpDet.tyLyr1.uiRtStat));
	END_IF

	//254 Characters are Shown
	IF tyP0400ProdSel.tyRcpDet.tyHotspotShowLRcp.bRtCompl = TRUE THEN
		tyP0400ProdSel.tyRcpDet.tyHotspotShowLRcp.bRtCompl  := FALSE;

		fUIInRtStatOff(ADR(tyP0400ProdSel.tyRcpPopUp.tyLyr.uiRtStat));

		tyP0400ProdSel.tyRcpPopUp.tyStringInfo.sValue  :=  tyP0400ProdSel.tyProdSel.tyTableRecipe.a_tyStringDataCol1[tyP0400Table.uiSelectedRow].sValue; // Show 254 Characters

	ELSIF tyP0400ProdSel.tyRcpPopUp.tyHotspotClose.bRtCompl = TRUE THEN
		tyP0400ProdSel.tyRcpPopUp.tyHotspotClose.bRtCompl := FALSE;

		fUIInRtStatHide(ADR(tyP0400ProdSel.tyRcpPopUp.tyLyr.uiRtStat)); // Hide Pop Up Again

	END_IF

END_ACTION
```

#### Act_EntP0410Disp.st
```iecst
ACTION Act_EntP0410Disp:

	//Access Addres
	IF p_tyNtParamCurr.eProjMag = LDMagQuadruple THEN
		p_tyC0004Navi ACCESS ADR(tyP0410MagSel.tyNavi2Lyr1);
	ELSIF p_tyNtParamCurr.eProjMag = LDMagTriple THEN
		p_tyC0004Navi ACCESS ADR(tyP0410MagSel.tyNavi1Lyr1);
	END_IF

	p_tyC0005Main ACCESS ADR(tyCommon.tyMain);

	p_tyC0007Notif ACCESS ADR(tyCommon.tyNotif);

	p_tyC0008MsgBox ACCESS ADR(tyP0410MagSel.tyMsgBoxHide);

	p_tyC0009Info ACCESS ADR(tyCommon.tyInfo);

	p_tyP0410MagSel ACCESS ADR(tyP0410MagSel.tyMagSel);

	p_tyP0410MagDet ACCESS ADR(tyP0410MagSel.tyMagDet);

	bRefreshMagRcpTable := TRUE;
	bMagazineRcpA := TRUE;
	bMagazineRcpB := FALSE;

	IF p_tyNtParamCurr.eProjMag = LDMagQuadruple THEN
		IF tyP0410MagSel.tyMagSel.tyTxtMagTitle.usiValueIdx	< 100 THEN
			tyP0410MagSel.tyMagSel.tyTxtMagTitle.usiValueIdx := tyP0410MagSel.tyMagSel.tyTxtMagTitle.usiValueIdx + 126;
		END_IF
	END_IF

	fUIInRtStatHide(ADR(tyP0410MagSel.tyMagDet.tyLyr.uiRtStat));

	// Enabling Display Auto Detect Magazine Mode
	tyP0410MagSel.tyMagSel.tyTxtMagModel.uiRtStat :=  NOT(p_tyNtParamCurr.bMagAutoVerifyPrep);

	tyP0410MagSel.tyMagSel.tyStringRecipeNm.sValue			:= p_tyMagRcpCurrRcp.sRcpNm;
	tyP0410MagSel.tyMagSel.tyNumSltToSltDist.diValue		:= p_tyMagRcpCurrRcp.diSltToSltInUM;
	tyP0410MagSel.tyMagSel.tyNumMaxSlt.diValue				:= p_tyMagRcpCurrRcp.diTtlSlt;
	tyP0410MagSel.tyMagSel.tyNumLifterMag1Slt1Pos.diValue	:= p_tyMagRcpCurrRcp.diMag1Slt1PosInUM;
	tyP0410MagSel.tyMagSel.tyNumLifterMag2Slt1Pos.diValue	:= p_tyMagRcpCurrRcp.diMag2Slt1PosInUM;
	tyP0410MagSel.tyMagSel.tyNumLifterMag3Slt1Pos.diValue	:= p_tyMagRcpCurrRcp.diMag3Slt1PosInUM;
	tyP0410MagSel.tyMagSel.tyNumLifterMag4Slt1Pos.diValue	:= p_tyMagRcpCurrRcp.diMag4Slt1PosInUM;
	tyP0410MagSel.tyMagSel.tyNumTravPosMag1.diValue			:= p_tyMagRcpCurrRcp.diMag1TravPosInUM;
	tyP0410MagSel.tyMagSel.tyNumTravPosMag2.diValue			:= p_tyMagRcpCurrRcp.diMag2TravPosInUM;
	tyP0410MagSel.tyMagSel.tyNumTravPosMag3.diValue			:= p_tyMagRcpCurrRcp.diMag3TravPosInUM;
	tyP0410MagSel.tyMagSel.tyNumTravPosMag4.diValue			:= p_tyMagRcpCurrRcp.diMag4TravPosInUM;
	tyP0410MagSel.tyMagSel.tyTxtMagModel.usiValueIdx		:= p_tyMagRcpCurrRcp.usiMagModel;
	tyP0410MagSel.tyMagSel.tyBtnSafetyBar.bValue			:= p_tyMagRcpCurrRcp.bSafetyBarDisabled;

END_ACTION
```
